LIN {X 0.059,Y -516.813,Z 888.156,A 0.000,B 0.000,C 90.000,E1 244.076} C_DIS
LIN {X -0.130,Y -514.887,Z 888.150,A 0.000,B 0.000,C 90.000,E1 242.922} C_DIS
LIN {X 0.096,Y -511.834,Z 888.140,A 0.000,B 0.000,C 90.000,E1 241.129} C_DIS
LIN {X -0.073,Y -508.198,Z 888.128,A 0.000,B 0.000,C 90.000,E1 239.076} C_DIS
LIN {X -0.008,Y -505.549,Z 888.120,A 0.000,B 0.000,C 90.000,E1 237.582} C_DIS
LIN {X 0.121,Y -503.196,Z 888.113,A 0.000,B 0.000,C 90.000,E1 236.373} C_DIS
LIN {X 0.071,Y -500.604,Z 888.107,A 0.000,B 0.000,C 90.000,E1 235.182} C_DIS
LIN {X -0.143,Y -497.089,Z 888.098,A 0.000,B 0.000,C 90.000,E1 233.703} C_DIS
LIN {X -0.267,Y -492.998,Z 888.088,A 0.000,B 0.000,C 90.000,E1 231.904} C_DIS
LIN {X -0.022,Y -489.498,Z 888.080,A 0.000,B 0.000,C 90.000,E1 230.356} C_DIS
LIN {X -0.047,Y -486.776,Z 888.073,A 0.000,B 0.000,C 90.000,E1 229.138} C_DIS
LIN {X 0.031,Y -483.298,Z 888.065,A 0.000,B 0.000,C 90.000,E1 227.595} C_DIS
LIN {X 0.037,Y -479.932,Z 888.056,A 0.000,B 0.000,C 90.000,E1 226.053} C_DIS
LIN {X 0.072,Y -475.754,Z 888.046,A 0.000,B 0.000,C 90.000,E1 224.190} C_DIS
LIN {X 0.120,Y -470.811,Z 888.033,A 0.000,B 0.000,C 90.000,E1 222.000} C_DIS
LIN {X -0.181,Y -468.009,Z 888.026,A 0.000,B 0.000,C 90.000,E1 220.782} C_DIS
LIN {X -0.109,Y -464.634,Z 888.018,A 0.000,B 0.000,C 90.000,E1 219.197} C_DIS
LIN {X -0.036,Y -461.259,Z 888.009,A 0.000,B 0.000,C 90.000,E1 217.604} C_DIS
LIN {X 0.078,Y -457.223,Z 887.998,A 0.000,B 0.000,C 90.000,E1 215.678} C_DIS
LIN {X -0.169,Y -453.164,Z 887.988,A 0.000,B 0.000,C 90.000,E1 213.785} C_DIS
LIN {X -0.069,Y -448.359,Z 887.975,A 0.000,B 0.000,C 90.000,E1 211.514} C_DIS
LIN {X 0.187,Y -443.374,Z 887.962,A 0.000,B 0.000,C 90.000,E1 209.205} C_DIS
LIN {X 0.179,Y -440.544,Z 887.955,A 0.000,B 0.000,C 90.000,E1 207.897} C_DIS
LIN {X -0.049,Y -436.846,Z 887.946,A 0.000,B 0.000,C 90.000,E1 206.283} C_DIS
LIN {X 0.072,Y -432.648,Z 887.935,A 0.000,B 0.000,C 90.000,E1 204.283} C_DIS
LIN {X 0.103,Y -428.359,Z 887.924,A 0.000,B 0.000,C 90.000,E1 202.280} C_DIS
LIN {X -0.126,Y -425.591,Z 887.916,A 0.000,B 0.000,C 90.000,E1 200.972} C_DIS
LIN {X -0.012,Y -420.825,Z 887.903,A 0.000,B 0.000,C 90.000,E1 198.598} C_DIS
LIN {X 0.069,Y -416.672,Z 887.892,A 0.000,B 0.000,C 90.000,E1 196.551} C_DIS
LIN {X -0.022,Y -411.180,Z 887.877,A 0.000,B 0.000,C 90.000,E1 193.828} C_DIS
LIN {X -0.115,Y -407.915,Z 887.867,A 0.000,B 0.000,C 90.000,E1 192.119} C_DIS
LIN {X 0.027,Y -405.234,Z 887.860,A 0.000,B 0.000,C 90.000,E1 190.715} C_DIS
LIN {X 0.043,Y -401.029,Z 887.848,A 0.000,B 0.000,C 90.000,E1 188.624} C_DIS
LIN {X -0.103,Y -396.837,Z 887.836,A 0.000,B 0.000,C 90.000,E1 186.543} C_DIS
LIN {X -0.116,Y -392.391,Z 887.823,A 0.000,B 0.000,C 90.000,E1 184.073} C_DIS
LIN {X -0.042,Y -387.473,Z 887.805,A 0.000,B 0.000,C 90.000,E1 180.859} C_DIS
LIN {X -0.040,Y -385.346,Z 887.797,A 0.000,B 0.000,C 90.000,E1 179.427} C_DIS
LIN {X -0.175,Y -382.648,Z 887.787,A 0.000,B 0.000,C 90.000,E1 177.650} C_DIS
LIN {X 0.135,Y -380.360,Z 887.779,A 0.000,B 0.000,C 90.000,E1 176.159} C_DIS
LIN {X -0.136,Y -376.095,Z 887.761,A 0.000,B 0.000,C 90.000,E1 172.932} C_DIS
LIN {X -0.027,Y -375.411,Z 887.757,A 0.000,B 0.000,C 90.000,E1 172.186} C_DIS
LIN {X 0.012,Y -374.903,Z 887.751,A 0.000,B 0.000,C 90.000,E1 171.084} C_DIS
LIN {X -0.099,Y -374.936,Z 887.748,A 0.000,B 0.000,C 90.000,E1 170.735} C_DIS
LIN {X 0.158,Y -374.805,Z 887.746,A 0.000,B 0.000,C 90.000,E1 170.330} C_DIS
LIN {X -0.090,Y -375.176,Z 887.741,A 0.000,B 0.000,C 90.000,E1 169.454} C_DIS
LIN {X 0.147,Y -375.812,Z 887.738,A 0.000,B 0.000,C 90.000,E1 168.870} C_DIS
LIN {X -0.001,Y -377.105,Z 887.734,A 0.000,B 0.000,C 90.000,E1 168.173} C_DIS
LIN {X -0.125,Y -378.598,Z 887.731,A 0.000,B 0.000,C 90.000,E1 167.645} C_DIS
LIN {X 0.093,Y -381.115,Z 887.728,A 0.000,B 0.000,C 90.000,E1 166.992} C_DIS
LIN {X -0.115,Y -384.469,Z 887.725,A 0.000,B 0.000,C 90.000,E1 166.464} C_DIS
LIN {X -0.114,Y -385.784,Z 887.724,A 0.000,B 0.000,C 90.000,E1 166.284} C_DIS
LIN {X 0.161,Y -389.176,Z 887.722,A 0.000,B 0.000,C 90.000,E1 165.880} C_DIS
LIN {X 0.093,Y -392.070,Z 887.720,A 0.000,B 0.000,C 90.000,E1 165.644} C_DIS
LIN {X 0.128,Y -398.264,Z 887.718,A 0.000,B 0.000,C 90.000,E1 165.227} C_DIS
LIN {X 0.093,Y -408.630,Z 887.715,A 0.000,B 0.000,C 90.000,E1 164.629} C_DIS
LIN {X -0.160,Y -413.785,Z 887.713,A 0.000,B 0.000,C 90.000,E1 164.393} C_DIS
LIN {X 0.051,Y -420.215,Z 887.711,A 0.000,B 0.000,C 90.000,E1 163.976} C_DIS
LIN {X -0.171,Y -429.850,Z 887.708,A 0.000,B 0.000,C 90.000,E1 163.378} C_DIS
LIN {X 0.016,Y -437.695,Z 887.704,A 0.000,B 0.000,C 90.000,E1 162.779} C_DIS
LIN {X 0.110,Y -446.755,Z 887.700,A 0.000,B 0.000,C 90.000,E1 162.000} C_DIS
LIN {X -0.047,Y -455.747,Z 887.696,A 0.000,B 0.000,C 90.000,E1 161.221} C_DIS
LIN {X 0.161,Y -464.336,Z 887.691,A 0.000,B 0.000,C 90.000,E1 160.369} C_DIS
LIN {X -0.030,Y -474.098,Z 887.686,A 0.000,B 0.000,C 90.000,E1 159.390} C_DIS
LIN {X 0.276,Y -481.913,Z 887.681,A 0.000,B 0.000,C 90.000,E1 158.465} C_DIS
LIN {X 0.065,Y -488.271,Z 887.676,A 0.000,B 0.000,C 90.000,E1 157.720} C_DIS
LIN {X 0.019,Y -499.849,Z 887.668,A 0.000,B 0.000,C 90.000,E1 156.230} C_DIS
LIN {X 0.044,Y -507.400,Z 887.662,A 0.000,B 0.000,C 90.000,E1 155.177} C_DIS
LIN {X 0.168,Y -510.575,Z 887.660,A 0.000,B 0.000,C 90.000,E1 154.717} C_DIS
LIN {X 0.050,Y -520.770,Z 887.651,A 0.000,B 0.000,C 90.000,E1 153.256} C_DIS
LIN {X -0.060,Y -528.491,Z 887.645,A 0.000,B 0.000,C 90.000,E1 152.103} C_DIS
LIN {X -0.099,Y -532.886,Z 887.641,A 0.000,B 0.000,C 90.000,E1 151.385} C_DIS
LIN {X -0.075,Y -538.842,Z 887.635,A 0.000,B 0.000,C 90.000,E1 150.383} C_DIS
LIN {X 0.117,Y -542.172,Z 887.632,A 0.000,B 0.000,C 90.000,E1 149.793} C_DIS
LIN {X -0.025,Y -549.222,Z 887.625,A 0.000,B 0.000,C 90.000,E1 148.535} C_DIS
LIN {X 0.188,Y -558.365,Z 887.616,A 0.000,B 0.000,C 90.000,E1 146.834} C_DIS
LIN {X 0.019,Y -565.388,Z 887.608,A 0.000,B 0.000,C 90.000,E1 145.468} C_DIS
LIN {X -0.177,Y -572.023,Z 887.601,A 0.000,B 0.000,C 90.000,E1 144.116} C_DIS
LIN {X 0.053,Y -577.218,Z 887.595,A 0.000,B 0.000,C 90.000,E1 143.004} C_DIS
LIN {X 0.242,Y -582.184,Z 887.589,A 0.000,B 0.000,C 90.000,E1 141.904} C_DIS
LIN {X -0.320,Y -587.103,Z 887.583,A 0.000,B 0.000,C 90.000,E1 140.884} C_DIS
LIN {X -0.248,Y -592.947,Z 887.575,A 0.000,B 0.000,C 90.000,E1 139.542} C_DIS
LIN {X 0.098,Y -599.979,Z 887.566,A 0.000,B 0.000,C 90.000,E1 137.919} C_DIS
LIN {X 0.146,Y -604.823,Z 887.560,A 0.000,B 0.000,C 90.000,E1 136.863} C_DIS
LIN {X -0.135,Y -611.955,Z 887.552,A 0.000,B 0.000,C 90.000,E1 135.324} C_DIS
LIN {X 0.051,Y -616.652,Z 887.546,A 0.000,B 0.000,C 90.000,E1 134.271} C_DIS
LIN {X -0.130,Y -621.125,Z 887.540,A 0.000,B 0.000,C 90.000,E1 133.257} C_DIS
LIN {X 0.311,Y -624.469,Z 887.536,A 0.000,B 0.000,C 90.000,E1 132.447} C_DIS
LIN {X -0.315,Y -629.897,Z 887.529,A 0.000,B 0.000,C 90.000,E1 131.229} C_DIS
LIN {X 0.152,Y -634.049,Z 887.523,A 0.000,B 0.000,C 90.000,E1 130.172} C_DIS
LIN {X -0.220,Y -638.094,Z 887.518,A 0.000,B 0.000,C 90.000,E1 129.197} C_DIS
LIN {X -0.147,Y -642.973,Z 887.511,A 0.000,B 0.000,C 90.000,E1 127.935} C_DIS
LIN {X 0.124,Y -647.825,Z 887.504,A 0.000,B 0.000,C 90.000,E1 126.664} C_DIS
LIN {X -0.044,Y -652.278,Z 887.497,A 0.000,B 0.000,C 90.000,E1 125.438} C_DIS
LIN {X 0.012,Y -656.493,Z 887.490,A 0.000,B 0.000,C 90.000,E1 124.199} C_DIS
LIN {X 0.144,Y -660.355,Z 887.483,A 0.000,B 0.000,C 90.000,E1 122.959} C_DIS
LIN {X 0.292,Y -662.401,Z 887.479,A 0.000,B 0.000,C 90.000,E1 122.212} C_DIS
LIN {X -0.105,Y -664.263,Z 887.475,A 0.000,B 0.000,C 90.000,E1 121.514} C_DIS
LIN {X -0.269,Y -665.852,Z 887.471,A 0.000,B 0.000,C 90.000,E1 120.797} C_DIS
LIN {X 0.075,Y -667.726,Z 887.466,A 0.000,B 0.000,C 90.000,E1 119.795} C_DIS
LIN {X -0.315,Y -669.714,Z 887.459,A 0.000,B 0.000,C 90.000,E1 118.615} C_DIS
LIN {X 0.256,Y -672.187,Z 887.449,A 0.000,B 0.000,C 90.000,E1 116.873} C_DIS
LIN {X 0.229,Y -673.346,Z 887.443,A 0.000,B 0.000,C 90.000,E1 115.668} C_DIS
LIN {X 0.150,Y -673.803,Z 887.439,A 0.000,B 0.000,C 90.000,E1 114.951} C_DIS
LIN {X -0.214,Y -674.045,Z 887.435,A 0.000,B 0.000,C 90.000,E1 114.259} C_DIS
LIN {X 0.041,Y -673.732,Z 887.431,A 0.000,B 0.000,C 90.000,E1 113.515} C_DIS
LIN {X 0.123,Y -672.857,Z 887.428,A 0.000,B 0.000,C 90.000,E1 113.025} C_DIS
LIN {X 0.294,Y -672.227,Z 887.427,A 0.000,B 0.000,C 90.000,E1 112.770} C_DIS
LIN {X -0.252,Y -669.397,Z 887.424,A 0.000,B 0.000,C 90.000,E1 112.333} C_DIS
LIN {X -0.172,Y -668.607,Z 887.423,A 0.000,B 0.000,C 90.000,E1 112.206} C_DIS
LIN {X -0.094,Y -667.531,Z 887.423,A 0.000,B 0.000,C 90.000,E1 112.078} C_DIS
LIN {X -0.171,Y -661.427,Z 887.420,A 0.000,B 0.000,C 90.000,E1 111.642} C_DIS
LIN {X -0.005,Y -659.918,Z 887.420,A 0.000,B 0.000,C 90.000,E1 111.535} C_DIS
LIN {X 0.346,Y -654.136,Z 887.418,A 0.000,B 0.000,C 90.000,E1 111.280} C_DIS
LIN {X 0.188,Y -652.034,Z 887.418,A 0.000,B 0.000,C 90.000,E1 111.227} C_DIS
LIN {X 0.362,Y -642.512,Z 887.417,A 0.000,B 0.000,C 90.000,E1 110.972} C_DIS
LIN {X -0.032,Y -634.972,Z 887.416,A 0.000,B 0.000,C 90.000,E1 110.844} C_DIS
LIN {X 0.254,Y -621.767,Z 887.414,A 0.000,B 0.000,C 90.000,E1 110.482} C_DIS
LIN {X 0.219,Y -615.744,Z 887.413,A 0.000,B 0.000,C 90.000,E1 110.301} C_DIS
LIN {X -0.145,Y -611.117,Z 887.412,A 0.000,B 0.000,C 90.000,E1 110.174} C_DIS
LIN {X 0.025,Y -603.066,Z 887.410,A 0.000,B 0.000,C 90.000,E1 109.812} C_DIS
LIN {X 0.054,Y -591.318,Z 887.407,A 0.000,B 0.000,C 90.000,E1 109.214} C_DIS
LIN {X 0.166,Y -588.091,Z 887.406,A 0.000,B 0.000,C 90.000,E1 109.033} C_DIS
LIN {X -0.159,Y -579.718,Z 887.404,A 0.000,B 0.000,C 90.000,E1 108.671} C_DIS
LIN {X -0.140,Y -567.602,Z 887.401,A 0.000,B 0.000,C 90.000,E1 108.236} C_DIS
LIN {X -0.094,Y -564.043,Z 887.401,A 0.000,B 0.000,C 90.000,E1 108.109} C_DIS
LIN {X 0.096,Y -562.050,Z 887.400,A 0.000,B 0.000,C 90.000,E1 108.000} C_DIS
LIN {X -0.011,Y -558.885,Z 887.399,A 0.000,B 0.000,C 90.000,E1 107.819} C_DIS
LIN {X -0.056,Y -558.823,Z 887.399,A 0.000,B 0.000,C 90.000,E1 107.819} C_DIS
LIN {X -0.160,Y -557.401,Z 887.398,A 0.000,B 0.000,C 90.000,E1 107.583} C_DIS
LIN {X -0.182,Y -556.754,Z 887.396,A 0.000,B 0.000,C 90.000,E1 107.221} C_DIS
LIN {X 0.149,Y -556.647,Z 887.391,A 0.000,B 0.000,C 90.000,E1 106.441} C_DIS
LIN {X 0.009,Y -557.505,Z 887.378,A 0.000,B 0.000,C 90.000,E1 103.953} C_DIS
LIN {X -0.235,Y -558.913,Z 887.364,A 0.000,B 0.000,C 90.000,E1 101.478} C_DIS
LIN {X 0.137,Y -560.336,Z 887.353,A 0.000,B 0.000,C 90.000,E1 99.500} C_DIS
LIN {X 0.239,Y -561.270,Z 887.345,A 0.000,B 0.000,C 90.000,E1 98.106} C_DIS
LIN {X -0.137,Y -562.309,Z 887.336,A 0.000,B 0.000,C 90.000,E1 96.486} C_DIS
LIN {X -0.237,Y -562.889,Z 887.330,A 0.000,B 0.000,C 90.000,E1 95.391} C_DIS
LIN {X -0.237,Y -563.548,Z 887.322,A 0.000,B 0.000,C 90.000,E1 94.012} C_DIS
LIN {X -0.261,Y -564.051,Z 887.315,A 0.000,B 0.000,C 90.000,E1 92.636} C_DIS
LIN {X -0.165,Y -564.603,Z 887.305,A 0.000,B 0.000,C 90.000,E1 90.974} C_DIS
LIN {X -0.067,Y -565.013,Z 887.296,A 0.000,B 0.000,C 90.000,E1 89.312} C_DIS
LIN {X -0.191,Y -565.269,Z 887.290,A 0.000,B 0.000,C 90.000,E1 88.224} C_DIS
LIN {X -0.156,Y -565.489,Z 887.282,A 0.000,B 0.000,C 90.000,E1 86.846} C_DIS
LIN {X 0.009,Y -565.757,Z 887.273,A 0.000,B 0.000,C 90.000,E1 85.179} C_DIS
LIN {X -0.142,Y -566.155,Z 887.261,A 0.000,B 0.000,C 90.000,E1 82.996} C_DIS
LIN {X -0.252,Y -566.636,Z 887.250,A 0.000,B 0.000,C 90.000,E1 81.084} C_DIS
LIN {X -0.249,Y -567.367,Z 887.240,A 0.000,B 0.000,C 90.000,E1 79.162} C_DIS
LIN {X -0.112,Y -568.261,Z 887.229,A 0.000,B 0.000,C 90.000,E1 77.229} C_DIS
LIN {X -0.006,Y -568.993,Z 887.220,A 0.000,B 0.000,C 90.000,E1 75.574} C_DIS
LIN {X 0.110,Y -569.714,Z 887.211,A 0.000,B 0.000,C 90.000,E1 73.921} C_DIS
LIN {X 0.179,Y -570.234,Z 887.200,A 0.000,B 0.000,C 90.000,E1 72.000} C_DIS
LIN {X -0.259,Y -570.502,Z 887.193,A 0.000,B 0.000,C 90.000,E1 70.678} C_DIS
LIN {X 0.059,Y -570.671,Z 887.188,A 0.000,B 0.000,C 90.000,E1 69.826} C_DIS
LIN {X -0.020,Y -570.836,Z 887.177,A 0.000,B 0.000,C 90.000,E1 67.922} C_DIS
LIN {X 0.167,Y -570.974,Z 887.170,A 0.000,B 0.000,C 90.000,E1 66.538} C_DIS
LIN {X -0.043,Y -570.967,Z 887.161,A 0.000,B 0.000,C 90.000,E1 64.921} C_DIS
LIN {X 0.227,Y -570.910,Z 887.152,A 0.000,B 0.000,C 90.000,E1 63.256} C_DIS
LIN {X -0.012,Y -570.603,Z 887.143,A 0.000,B 0.000,C 90.000,E1 61.641} C_DIS
LIN {X 0.187,Y -570.303,Z 887.135,A 0.000,B 0.000,C 90.000,E1 60.255} C_DIS
LIN {X -0.160,Y -570.175,Z 887.132,A 0.000,B 0.000,C 90.000,E1 59.744} C_DIS
LIN {X 0.134,Y -569.278,Z 887.123,A 0.000,B 0.000,C 90.000,E1 58.074} C_DIS
LIN {X 0.065,Y -569.010,Z 887.120,A 0.000,B 0.000,C 90.000,E1 57.533} C_DIS
LIN {X 0.233,Y -568.153,Z 887.114,A 0.000,B 0.000,C 90.000,E1 56.421} C_DIS
LIN {X 0.072,Y -567.176,Z 887.108,A 0.000,B 0.000,C 90.000,E1 55.341} C_DIS
LIN {X -0.249,Y -566.038,Z 887.101,A 0.000,B 0.000,C 90.000,E1 54.276} C_DIS
LIN {X 0.209,Y -564.558,Z 887.095,A 0.000,B 0.000,C 90.000,E1 53.130} C_DIS
LIN {X 0.091,Y -563.392,Z 887.091,A 0.000,B 0.000,C 90.000,E1 52.316} C_DIS
LIN {X 0.059,Y -562.076,Z 887.086,A 0.000,B 0.000,C 90.000,E1 51.492} C_DIS
LIN {X -0.086,Y -560.550,Z 887.082,A 0.000,B 0.000,C 90.000,E1 50.678} C_DIS
LIN {X 0.114,Y -558.831,Z 887.077,A 0.000,B 0.000,C 90.000,E1 49.828} C_DIS
LIN {X -0.141,Y -557.534,Z 887.074,A 0.000,B 0.000,C 90.000,E1 49.299} C_DIS
LIN {X 0.036,Y -555.312,Z 887.069,A 0.000,B 0.000,C 90.000,E1 48.447} C_DIS
LIN {X -0.181,Y -552.730,Z 887.065,A 0.000,B 0.000,C 90.000,E1 47.634} C_DIS
LIN {X -0.059,Y -549.844,Z 887.060,A 0.000,B 0.000,C 90.000,E1 46.782} C_DIS
LIN {X -0.365,Y -546.736,Z 887.055,A 0.000,B 0.000,C 90.000,E1 45.972} C_DIS
LIN {X 0.061,Y -544.472,Z 887.052,A 0.000,B 0.000,C 90.000,E1 45.364} C_DIS
LIN {X 0.268,Y -542.728,Z 887.050,A 0.000,B 0.000,C 90.000,E1 44.919} C_DIS
LIN {X -0.302,Y -539.400,Z 887.046,A 0.000,B 0.000,C 90.000,E1 44.271} C_DIS
LIN {X 0.067,Y -536.531,Z 887.043,A 0.000,B 0.000,C 90.000,E1 43.662} C_DIS
LIN {X 0.200,Y -532.521,Z 887.039,A 0.000,B 0.000,C 90.000,E1 42.933} C_DIS
LIN {X -0.064,Y -528.181,Z 887.035,A 0.000,B 0.000,C 90.000,E1 42.243} C_DIS
LIN {X -0.211,Y -522.699,Z 887.030,A 0.000,B 0.000,C 90.000,E1 41.391} C_DIS
LIN {X 0.111,Y -515.454,Z 887.024,A 0.000,B 0.000,C 90.000,E1 40.334} C_DIS
LIN {X -0.300,Y -509.888,Z 887.020,A 0.000,B 0.000,C 90.000,E1 39.644} C_DIS
LIN {X -0.051,Y -503.734,Z 887.016,A 0.000,B 0.000,C 90.000,E1 38.874} C_DIS
LIN {X 0.023,Y -499.850,Z 887.013,A 0.000,B 0.000,C 90.000,E1 38.418} C_DIS
LIN {X 0.121,Y -495.848,Z 887.011,A 0.000,B 0.000,C 90.000,E1 37.971} C_DIS
LIN {X -0.254,Y -490.285,Z 887.008,A 0.000,B 0.000,C 90.000,E1 37.443} C_DIS
LIN {X 0.038,Y -483.201,Z 887.004,A 0.000,B 0.000,C 90.000,E1 36.710} C_DIS
LIN {X 0.255,Y -475.862,Z 887.000,A 0.000,B 0.000,C 90.000,E1 36.011} C_DIS
LIN {X -0.122,Y -465.301,Z 886.995,A 0.000,B 0.000,C 90.000,E1 35.152} C_DIS
LIN {X -0.131,Y -454.806,Z 886.990,A 0.000,B 0.000,C 90.000,E1 34.278} C_DIS
LIN {X 0.057,Y -437.675,Z 886.983,A 0.000,B 0.000,C 90.000,E1 32.880} C_DIS
LIN {X 0.055,Y -416.158,Z 886.973,A 0.000,B 0.000,C 90.000,E1 31.052} C_DIS
LIN {X -0.042,Y -402.686,Z 886.966,A 0.000,B 0.000,C 90.000,E1 29.795} C_DIS
LIN {X 0.018,Y -398.395,Z 886.963,A 0.000,B 0.000,C 90.000,E1 29.333} C_DIS
LIN {X -0.224,Y -394.895,Z 886.961,A 0.000,B 0.000,C 90.000,E1 28.949} C_DIS
LIN {X -0.097,Y -391.850,Z 886.958,A 0.000,B 0.000,C 90.000,E1 28.409} C_DIS
LIN {X 0.110,Y -390.090,Z 886.955,A 0.000,B 0.000,C 90.000,E1 27.847} C_DIS
LIN {X 0.148,Y -389.174,Z 886.951,A 0.000,B 0.000,C 90.000,E1 27.129} C_DIS
LIN {X 0.182,Y -389.082,Z 886.946,A 0.000,B 0.000,C 90.000,E1 26.232} C_DIS
LIN {X 0.056,Y -389.793,Z 886.938,A 0.000,B 0.000,C 90.000,E1 24.823} C_DIS
LIN {X 0.036,Y -391.867,Z 886.924,A 0.000,B 0.000,C 90.000,E1 22.333} C_DIS
LIN {X -0.018,Y -394.747,Z 886.908,A 0.000,B 0.000,C 90.000,E1 19.504} C_DIS
LIN {X -0.067,Y -397.577,Z 886.895,A 0.000,B 0.000,C 90.000,E1 17.040} C_DIS
LIN {X -0.150,Y -400.720,Z 886.881,A 0.000,B 0.000,C 90.000,E1 14.592} C_DIS
LIN {X 0.038,Y -405.029,Z 886.864,A 0.000,B 0.000,C 90.000,E1 11.422} C_DIS
LIN {X 0.158,Y -407.697,Z 886.854,A 0.000,B 0.000,C 90.000,E1 9.670} C_DIS
LIN {X -0.155,Y -411.645,Z 886.840,A 0.000,B 0.000,C 90.000,E1 7.296} C_DIS
LIN {X 0.000,Y -416.709,Z 886.825,A 0.000,B 0.000,C 90.000,E1 4.531} C_DIS
LIN {X -0.089,Y -423.732,Z 886.806,A 0.000,B 0.000,C 90.000,E1 1.146} C_DIS
LIN {X -0.081,Y -429.251,Z 886.793,A 0.000,B 0.000,C 90.000,E1 358.797} C_DIS
LIN {X 0.145,Y -436.063,Z 886.779,A 0.000,B 0.000,C 90.000,E1 356.102} C_DIS
LIN {X -0.077,Y -438.183,Z 886.775,A 0.000,B 0.000,C 90.000,E1 355.469} C_DIS
LIN {X 0.055,Y -439.675,Z 886.773,A 0.000,B 0.000,C 90.000,E1 355.122} C_DIS
LIN {X 0.001,Y -442.807,Z 886.770,A 0.000,B 0.000,C 90.000,E1 354.609} C_DIS
LIN {X -0.192,Y -443.523,Z 886.770,A 0.000,B 0.000,C 90.000,E1 354.546} C_DIS
LIN {X 0.015,Y -444.471,Z 886.769,A 0.000,B 0.000,C 90.000,E1 354.432} C_DIS
LIN {X -0.016,Y -449.205,Z 886.767,A 0.000,B 0.000,C 90.000,E1 354.090} C_DIS
LIN {X 0.103,Y -456.288,Z 886.765,A 0.000,B 0.000,C 90.000,E1 353.742} C_DIS
LIN {X -0.076,Y -468.575,Z 886.762,A 0.000,B 0.000,C 90.000,E1 353.223} C_DIS
LIN {X 0.223,Y -475.053,Z 886.761,A 0.000,B 0.000,C 90.000,E1 352.875} C_DIS
LIN {X 0.208,Y -481.798,Z 886.759,A 0.000,B 0.000,C 90.000,E1 352.534} C_DIS
LIN {X 0.135,Y -491.540,Z 886.756,A 0.000,B 0.000,C 90.000,E1 352.008} C_DIS
LIN {X 0.171,Y -501.419,Z 886.753,A 0.000,B 0.000,C 90.000,E1 351.432} C_DIS
LIN {X -0.122,Y -513.963,Z 886.748,A 0.000,B 0.000,C 90.000,E1 350.679} C_DIS
LIN {X -0.079,Y -521.715,Z 886.745,A 0.000,B 0.000,C 90.000,E1 350.151} C_DIS
LIN {X 0.198,Y -529.264,Z 886.742,A 0.000,B 0.000,C 90.000,E1 349.577} C_DIS
LIN {X -0.223,Y -538.117,Z 886.738,A 0.000,B 0.000,C 90.000,E1 348.926} C_DIS
LIN {X 0.153,Y -543.635,Z 886.736,A 0.000,B 0.000,C 90.000,E1 348.409} C_DIS
LIN {X -0.136,Y -549.131,Z 886.733,A 0.000,B 0.000,C 90.000,E1 347.937} C_DIS
LIN {X -0.033,Y -554.512,Z 886.730,A 0.000,B 0.000,C 90.000,E1 347.409} C_DIS
LIN {X -0.159,Y -560.835,Z 886.726,A 0.000,B 0.000,C 90.000,E1 346.756} C_DIS
LIN {X -0.069,Y -566.929,Z 886.723,A 0.000,B 0.000,C 90.000,E1 346.061} C_DIS
LIN {X -0.139,Y -571.537,Z 886.720,A 0.000,B 0.000,C 90.000,E1 345.519} C_DIS
LIN {X -0.121,Y -577.964,Z 886.715,A 0.000,B 0.000,C 90.000,E1 344.700} C_DIS
LIN {X 0.114,Y -583.849,Z 886.710,A 0.000,B 0.000,C 90.000,E1 343.866} C_DIS
LIN {X -0.150,Y -589.341,Z 886.706,A 0.000,B 0.000,C 90.000,E1 343.087} C_DIS
LIN {X 0.021,Y -596.755,Z 886.699,A 0.000,B 0.000,C 90.000,E1 341.873} C_DIS
LIN {X -0.111,Y -601.276,Z 886.695,A 0.000,B 0.000,C 90.000,E1 341.094} C_DIS
LIN {X -0.247,Y -606.318,Z 886.690,A 0.000,B 0.000,C 90.000,E1 340.188} C_DIS
LIN {X -0.384,Y -612.346,Z 886.683,A 0.000,B 0.000,C 90.000,E1 339.028} C_DIS
LIN {X -0.178,Y -616.855,Z 886.678,A 0.000,B 0.000,C 90.000,E1 338.103} C_DIS
LIN {X 0.078,Y -621.677,Z 886.673,A 0.000,B 0.000,C 90.000,E1 337.050} C_DIS
LIN {X -0.181,Y -626.221,Z 886.667,A 0.000,B 0.000,C 90.000,E1 336.049} C_DIS
LIN {X -0.120,Y -630.452,Z 886.661,A 0.000,B 0.000,C 90.000,E1 335.025} C_DIS
LIN {X -0.267,Y -634.393,Z 886.656,A 0.000,B 0.000,C 90.000,E1 334.024} C_DIS
LIN {X -0.090,Y -638.035,Z 886.650,A 0.000,B 0.000,C 90.000,E1 332.999} C_DIS
LIN {X 0.017,Y -639.804,Z 886.647,A 0.000,B 0.000,C 90.000,E1 332.487} C_DIS
LIN {X -0.303,Y -643.095,Z 886.642,A 0.000,B 0.000,C 90.000,E1 331.513} C_DIS
LIN {X 0.295,Y -646.090,Z 886.636,A 0.000,B 0.000,C 90.000,E1 330.461} C_DIS
LIN {X 0.048,Y -649.045,Z 886.631,A 0.000,B 0.000,C 90.000,E1 329.488} C_DIS
LIN {X 0.039,Y -652.487,Z 886.624,A 0.000,B 0.000,C 90.000,E1 328.250} C_DIS
LIN {X -0.241,Y -654.411,Z 886.620,A 0.000,B 0.000,C 90.000,E1 327.533} C_DIS
LIN {X -0.155,Y -657.153,Z 886.613,A 0.000,B 0.000,C 90.000,E1 326.294} C_DIS
LIN {X -0.119,Y -659.133,Z 886.607,A 0.000,B 0.000,C 90.000,E1 325.308} C_DIS
LIN {X 0.042,Y -661.153,Z 886.600,A 0.000,B 0.000,C 90.000,E1 324.069} C_DIS
LIN {X -0.404,Y -662.539,Z 886.595,A 0.000,B 0.000,C 90.000,E1 323.130} C_DIS
LIN {X 0.102,Y -663.796,Z 886.590,A 0.000,B 0.000,C 90.000,E1 322.110} C_DIS
LIN {X 0.188,Y -665.124,Z 886.583,A 0.000,B 0.000,C 90.000,E1 320.884} C_DIS
LIN {X 0.249,Y -667.167,Z 886.572,A 0.000,B 0.000,C 90.000,E1 318.933} C_DIS
LIN {X 0.302,Y -668.974,Z 886.563,A 0.000,B 0.000,C 90.000,E1 317.229} C_DIS
LIN {X -0.104,Y -670.500,Z 886.555,A 0.000,B 0.000,C 90.000,E1 315.810} C_DIS
LIN {X -0.015,Y -671.971,Z 886.546,A 0.000,B 0.000,C 90.000,E1 314.352} C_DIS
LIN {X -0.324,Y -673.867,Z 886.536,A 0.000,B 0.000,C 90.000,E1 312.447} C_DIS
LIN {X -0.168,Y -674.987,Z 886.529,A 0.000,B 0.000,C 90.000,E1 311.229} C_DIS
LIN {X 0.155,Y -676.657,Z 886.518,A 0.000,B 0.000,C 90.000,E1 309.277} C_DIS
LIN {X -0.078,Y -677.578,Z 886.512,A 0.000,B 0.000,C 90.000,E1 308.096} C_DIS
LIN {X 0.235,Y -678.498,Z 886.505,A 0.000,B 0.000,C 90.000,E1 306.870} C_DIS
LIN {X 0.164,Y -679.304,Z 886.498,A 0.000,B 0.000,C 90.000,E1 305.678} C_DIS
LIN {X 0.108,Y -680.035,Z 886.492,A 0.000,B 0.000,C 90.000,E1 304.485} C_DIS
LIN {X 0.409,Y -681.239,Z 886.481,A 0.000,B 0.000,C 90.000,E1 302.546} C_DIS
LIN {X 0.004,Y -682.660,Z 886.470,A 0.000,B 0.000,C 90.000,E1 300.669} C_DIS
LIN {X 0.009,Y -684.099,Z 886.461,A 0.000,B 0.000,C 90.000,E1 298.999} C_DIS
LIN {X 0.211,Y -686.165,Z 886.451,A 0.000,B 0.000,C 90.000,E1 297.078} C_DIS
LIN {X -0.142,Y -688.455,Z 886.440,A 0.000,B 0.000,C 90.000,E1 295.207} C_DIS
LIN {X -0.194,Y -689.561,Z 886.433,A 0.000,B 0.000,C 90.000,E1 294.027} C_DIS
LIN {X 0.268,Y -689.916,Z 886.431,A 0.000,B 0.000,C 90.000,E1 293.515} C_DIS
LIN {X -0.408,Y -689.929,Z 886.430,A 0.000,B 0.000,C 90.000,E1 293.334} C_DIS
LIN {X 0.051,Y -689.678,Z 886.427,A 0.000,B 0.000,C 90.000,E1 292.823} C_DIS
LIN {X 0.013,Y -689.142,Z 886.426,A 0.000,B 0.000,C 90.000,E1 292.589} C_DIS
LIN {X 0.204,Y -687.622,Z 886.423,A 0.000,B 0.000,C 90.000,E1 292.099} C_DIS
LIN {X -0.323,Y -686.971,Z 886.422,A 0.000,B 0.000,C 90.000,E1 292.025} C_DIS
LIN {X -0.212,Y -685.996,Z 886.422,A 0.000,B 0.000,C 90.000,E1 291.897} C_DIS
LIN {X 0.001,Y -683.493,Z 886.420,A 0.000,B 0.000,C 90.000,E1 291.642} C_DIS
LIN {X 0.104,Y -680.957,Z 886.419,A 0.000,B 0.000,C 90.000,E1 291.408} C_DIS
LIN {X 0.282,Y -679.253,Z 886.418,A 0.000,B 0.000,C 90.000,E1 291.280} C_DIS
LIN {X 0.213,Y -676.257,Z 886.418,A 0.000,B 0.000,C 90.000,E1 291.173} C_DIS
LIN {X -0.184,Y -669.080,Z 886.416,A 0.000,B 0.000,C 90.000,E1 290.972} C_DIS
LIN {X 0.061,Y -661.537,Z 886.415,A 0.000,B 0.000,C 90.000,E1 290.737} C_DIS
LIN {X -0.183,Y -656.899,Z 886.414,A 0.000,B 0.000,C 90.000,E1 290.536} C_DIS
LIN {X 0.374,Y -656.815,Z 886.414,A 0.000,B 0.000,C 90.000,E1 290.482} C_DIS
LIN {X -0.016,Y -655.833,Z 886.413,A 0.000,B 0.000,C 90.000,E1 290.375} C_DIS
LIN {X -0.060,Y -655.822,Z 886.413,A 0.000,B 0.000,C 90.000,E1 290.375} C_DIS
LIN {X -0.046,Y -655.737,Z 886.412,A 0.000,B 0.000,C 90.000,E1 290.174} C_DIS
LIN {X -0.077,Y -657.252,Z 886.409,A 0.000,B 0.000,C 90.000,E1 289.685} C_DIS
LIN {X -0.209,Y -660.425,Z 886.406,A 0.000,B 0.000,C 90.000,E1 289.033} C_DIS
LIN {X -0.201,Y -664.986,Z 886.401,A 0.000,B 0.000,C 90.000,E1 288.181} C_DIS
LIN {X -0.236,Y -666.887,Z 886.399,A 0.000,B 0.000,C 90.000,E1 287.819} C_DIS
LIN {X -0.285,Y -670.305,Z 886.395,A 0.000,B 0.000,C 90.000,E1 287.094} C_DIS
LIN {X 0.214,Y -672.292,Z 886.392,A 0.000,B 0.000,C 90.000,E1 286.567} C_DIS
LIN {X 0.216,Y -674.817,Z 886.388,A 0.000,B 0.000,C 90.000,E1 285.843} C_DIS
LIN {X 0.055,Y -676.701,Z 886.384,A 0.000,B 0.000,C 90.000,E1 285.134} C_DIS
LIN {X -0.040,Y -677.804,Z 886.381,A 0.000,B 0.000,C 90.000,E1 284.662} C_DIS
LIN {X -0.004,Y -679.141,Z 886.378,A 0.000,B 0.000,C 90.000,E1 283.939} C_DIS
LIN {X -0.282,Y -680.271,Z 886.373,A 0.000,B 0.000,C 90.000,E1 283.244} C_DIS
LIN {X 0.276,Y -681.127,Z 886.370,A 0.000,B 0.000,C 90.000,E1 282.479} C_DIS
LIN {X 0.173,Y -681.667,Z 886.366,A 0.000,B 0.000,C 90.000,E1 281.771} C_DIS
LIN {X 0.103,Y -681.830,Z 886.363,A 0.000,B 0.000,C 90.000,E1 281.299} C_DIS
LIN {X -0.133,Y -681.447,Z 886.359,A 0.000,B 0.000,C 90.000,E1 280.602} C_DIS
LIN {X -0.330,Y -680.970,Z 886.356,A 0.000,B 0.000,C 90.000,E1 280.141} C_DIS
LIN {X 0.261,Y -680.172,Z 886.354,A 0.000,B 0.000,C 90.000,E1 279.613} C_DIS
LIN {X 0.060,Y -679.042,Z 886.351,A 0.000,B 0.000,C 90.000,E1 279.151} C_DIS
LIN {X -0.195,Y -676.772,Z 886.347,A 0.000,B 0.000,C 90.000,E1 278.454} C_DIS
LIN {X 0.259,Y -674.965,Z 886.344,A 0.000,B 0.000,C 90.000,E1 277.936} C_DIS
LIN {X 0.035,Y -672.807,Z 886.342,A 0.000,B 0.000,C 90.000,E1 277.473} C_DIS
LIN {X -0.201,Y -669.739,Z 886.338,A 0.000,B 0.000,C 90.000,E1 276.891} C_DIS
LIN {X 0.116,Y -666.230,Z 886.335,A 0.000,B 0.000,C 90.000,E1 276.258} C_DIS
LIN {X -0.167,Y -663.120,Z 886.332,A 0.000,B 0.000,C 90.000,E1 275.796} C_DIS
LIN {X 0.186,Y -659.553,Z 886.329,A 0.000,B 0.000,C 90.000,E1 275.277} C_DIS
LIN {X -0.196,Y -655.508,Z 886.327,A 0.000,B 0.000,C 90.000,E1 274.821} C_DIS
LIN {X 0.134,Y -649.860,Z 886.323,A 0.000,B 0.000,C 90.000,E1 274.188} C_DIS
LIN {X -0.004,Y -645.037,Z 886.321,A 0.000,B 0.000,C 90.000,E1 273.726} C_DIS
LIN {X -0.144,Y -638.427,Z 886.318,A 0.000,B 0.000,C 90.000,E1 273.154} C_DIS
LIN {X 0.024,Y -631.476,Z 886.314,A 0.000,B 0.000,C 90.000,E1 272.579} C_DIS
LIN {X -0.023,Y -623.963,Z 886.312,A 0.000,B 0.000,C 90.000,E1 272.064} C_DIS
LIN {X 0.152,Y -617.581,Z 886.309,A 0.000,B 0.000,C 90.000,E1 271.661} C_DIS
LIN {X 0.008,Y -611.071,Z 886.307,A 0.000,B 0.000,C 90.000,E1 271.318} C_DIS
LIN {X 0.093,Y -602.622,Z 886.305,A 0.000,B 0.000,C 90.000,E1 270.917} C_DIS
LIN {X 0.192,Y -597.525,Z 886.304,A 0.000,B 0.000,C 90.000,E1 270.688} C_DIS
LIN {X -0.232,Y -589.970,Z 886.302,A 0.000,B 0.000,C 90.000,E1 270.458} C_DIS
LIN {X -0.244,Y -584.419,Z 886.302,A 0.000,B 0.000,C 90.000,E1 270.286} C_DIS
LIN {X 0.062,Y -576.820,Z 886.300,A 0.000,B 0.000,C 90.000,E1 270.057} C_DIS
LIN {X 0.026,Y -570.829,Z 886.300,A 0.000,B 0.000,C 90.000,E1 269.943} C_DIS
LIN {X -0.119,Y -564.792,Z 886.299,A 0.000,B 0.000,C 90.000,E1 269.885} C_DIS
LIN {X 0.045,Y -552.116,Z 886.299,A 0.000,B 0.000,C 90.000,E1 269.771} C_DIS
LIN {X -0.037,Y -549.913,Z 886.298,A 0.000,B 0.000,C 90.000,E1 269.714} C_DIS
LIN {X -0.080,Y -549.791,Z 886.298,A 0.000,B 0.000,C 90.000,E1 269.714} C_DIS
LIN {X 0.052,Y -548.303,Z 886.298,A 0.000,B 0.000,C 90.000,E1 269.542} C_DIS
LIN {X 0.013,Y -546.367,Z 886.297,A 0.000,B 0.000,C 90.000,E1 269.370} C_DIS
LIN {X -0.026,Y -546.334,Z 886.297,A 0.000,B 0.000,C 90.000,E1 269.370} C_DIS
LIN {X 0.161,Y -545.150,Z 886.294,A 0.000,B 0.000,C 90.000,E1 268.854} C_DIS
LIN {X -0.137,Y -543.395,Z 886.286,A 0.000,B 0.000,C 90.000,E1 267.478} C_DIS
LIN {X 0.197,Y -541.262,Z 886.270,A 0.000,B 0.000,C 90.000,E1 264.609} C_DIS
LIN {X -0.130,Y -540.337,Z 886.262,A 0.000,B 0.000,C 90.000,E1 263.223} C_DIS
LIN {X 0.072,Y -539.410,Z 886.256,A 0.000,B 0.000,C 90.000,E1 262.064} C_DIS
LIN {X -0.287,Y -538.034,Z 886.248,A 0.000,B 0.000,C 90.000,E1 260.679} C_DIS
LIN {X 0.156,Y -535.947,Z 886.237,A 0.000,B 0.000,C 90.000,E1 258.634} C_DIS
LIN {X -0.081,Y -534.405,Z 886.229,A 0.000,B 0.000,C 90.000,E1 257.229} C_DIS
LIN {X -0.181,Y -532.235,Z 886.219,A 0.000,B 0.000,C 90.000,E1 255.519} C_DIS
LIN {X -0.195,Y -530.058,Z 886.210,A 0.000,B 0.000,C 90.000,E1 253.795} C_DIS
LIN {X -0.106,Y -528.026,Z 886.200,A 0.000,B 0.000,C 90.000,E1 252.054} C_DIS
LIN {X 0.083,Y -526.906,Z 886.195,A 0.000,B 0.000,C 90.000,E1 251.167} C_DIS
LIN {X -0.061,Y -524.711,Z 886.186,A 0.000,B 0.000,C 90.000,E1 249.444} C_DIS
LIN {X -0.075,Y -523.132,Z 886.179,A 0.000,B 0.000,C 90.000,E1 248.284} C_DIS
LIN {X 0.233,Y -521.027,Z 886.171,A 0.000,B 0.000,C 90.000,E1 246.794} C_DIS
LIN {X -0.121,Y -519.243,Z 886.165,A 0.000,B 0.000,C 90.000,E1 245.665} C_DIS
LIN {X -0.144,Y -517.037,Z 886.157,A 0.000,B 0.000,C 90.000,E1 244.204} C_DIS
LIN {X 0.007,Y -515.611,Z 886.152,A 0.000,B 0.000,C 90.000,E1 243.307} C_DIS
LIN {X -0.093,Y -513.057,Z 886.144,A 0.000,B 0.000,C 90.000,E1 241.847} C_DIS
LIN {X -0.105,Y -511.014,Z 886.137,A 0.000,B 0.000,C 90.000,E1 240.667} C_DIS
LIN {X -0.255,Y -508.458,Z 886.129,A 0.000,B 0.000,C 90.000,E1 239.203} C_DIS
LIN {X -0.076,Y -506.301,Z 886.122,A 0.000,B 0.000,C 90.000,E1 237.995} C_DIS
LIN {X -0.245,Y -504.636,Z 886.117,A 0.000,B 0.000,C 90.000,E1 237.120} C_DIS
LIN {X 0.028,Y -501.586,Z 886.109,A 0.000,B 0.000,C 90.000,E1 235.595} C_DIS
LIN {X -0.040,Y -498.826,Z 886.102,A 0.000,B 0.000,C 90.000,E1 234.402} C_DIS
LIN {X 0.270,Y -494.676,Z 886.092,A 0.000,B 0.000,C 90.000,E1 232.557} C_DIS
LIN {X -0.299,Y -490.500,Z 886.082,A 0.000,B 0.000,C 90.000,E1 230.803} C_DIS
LIN {X 0.040,Y -486.313,Z 886.072,A 0.000,B 0.000,C 90.000,E1 228.933} C_DIS
LIN {X -0.036,Y -483.549,Z 886.065,A 0.000,B 0.000,C 90.000,E1 227.715} C_DIS
LIN {X 0.299,Y -480.210,Z 886.057,A 0.000,B 0.000,C 90.000,E1 226.134} C_DIS
LIN {X -0.002,Y -476.069,Z 886.046,A 0.000,B 0.000,C 90.000,E1 224.312} C_DIS
LIN {X -0.187,Y -470.438,Z 886.032,A 0.000,B 0.000,C 90.000,E1 221.838} C_DIS
LIN {X 0.172,Y -464.930,Z 886.018,A 0.000,B 0.000,C 90.000,E1 219.277} C_DIS
LIN {X 0.000,Y -460.827,Z 886.008,A 0.000,B 0.000,C 90.000,E1 217.397} C_DIS
LIN {X 0.000,Y -457.518,Z 885.999,A 0.000,B 0.000,C 90.000,E1 215.804} C_DIS
LIN {X 0.132,Y -453.464,Z 885.988,A 0.000,B 0.000,C 90.000,E1 213.865} C_DIS
LIN {X 0.243,Y -448.641,Z 885.976,A 0.000,B 0.000,C 90.000,E1 211.592} C_DIS
LIN {X 0.062,Y -444.389,Z 885.965,A 0.000,B 0.000,C 90.000,E1 209.667} C_DIS
LIN {X 0.072,Y -441.636,Z 885.958,A 0.000,B 0.000,C 90.000,E1 208.359} C_DIS
LIN {X -0.129,Y -437.912,Z 885.949,A 0.000,B 0.000,C 90.000,E1 206.744} C_DIS
LIN {X 0.206,Y -432.995,Z 885.936,A 0.000,B 0.000,C 90.000,E1 204.387} C_DIS
LIN {X 0.069,Y -428.701,Z 885.925,A 0.000,B 0.000,C 90.000,E1 202.408} C_DIS
LIN {X 0.044,Y -425.230,Z 885.915,A 0.000,B 0.000,C 90.000,E1 200.737} C_DIS
LIN {X -0.023,Y -421.196,Z 885.904,A 0.000,B 0.000,C 90.000,E1 198.725} C_DIS
LIN {X 0.070,Y -417.026,Z 885.893,A 0.000,B 0.000,C 90.000,E1 196.677} C_DIS
LIN {X 0.000,Y -411.536,Z 885.878,A 0.000,B 0.000,C 90.000,E1 193.953} C_DIS
LIN {X 0.026,Y -407.599,Z 885.866,A 0.000,B 0.000,C 90.000,E1 191.883} C_DIS
LIN {X 0.085,Y -404.887,Z 885.858,A 0.000,B 0.000,C 90.000,E1 190.489} C_DIS
LIN {X 0.106,Y -401.408,Z 885.849,A 0.000,B 0.000,C 90.000,E1 188.746} C_DIS
LIN {X -0.020,Y -397.193,Z 885.837,A 0.000,B 0.000,C 90.000,E1 186.663} C_DIS
LIN {X -0.033,Y -392.114,Z 885.821,A 0.000,B 0.000,C 90.000,E1 183.841} C_DIS
LIN {X 0.008,Y -387.312,Z 885.804,A 0.000,B 0.000,C 90.000,E1 180.630} C_DIS
LIN {X 0.006,Y -385.134,Z 885.796,A 0.000,B 0.000,C 90.000,E1 179.198} C_DIS
LIN {X -0.134,Y -382.474,Z 885.786,A 0.000,B 0.000,C 90.000,E1 177.421} C_DIS
LIN {X -0.085,Y -380.779,Z 885.780,A 0.000,B 0.000,C 90.000,E1 176.331} C_DIS
LIN {X 0.152,Y -375.555,Z 885.757,A 0.000,B 0.000,C 90.000,E1 172.299} C_DIS
LIN {X 0.195,Y -374.826,Z 885.751,A 0.000,B 0.000,C 90.000,E1 171.197} C_DIS
LIN {X -0.028,Y -374.622,Z 885.747,A 0.000,B 0.000,C 90.000,E1 170.500} C_DIS
LIN {X 0.026,Y -374.697,Z 885.742,A 0.000,B 0.000,C 90.000,E1 169.577} C_DIS
LIN {X -0.074,Y -375.104,Z 885.740,A 0.000,B 0.000,C 90.000,E1 169.162} C_DIS
LIN {X 0.067,Y -375.648,Z 885.736,A 0.000,B 0.000,C 90.000,E1 168.409} C_DIS
LIN {X -0.080,Y -377.174,Z 885.732,A 0.000,B 0.000,C 90.000,E1 167.701} C_DIS
LIN {X 0.167,Y -378.930,Z 885.729,A 0.000,B 0.000,C 90.000,E1 167.117} C_DIS
LIN {X 0.054,Y -381.129,Z 885.726,A 0.000,B 0.000,C 90.000,E1 166.589} C_DIS
LIN {X -0.046,Y -384.164,Z 885.723,A 0.000,B 0.000,C 90.000,E1 166.061} C_DIS
LIN {X 0.008,Y -387.061,Z 885.721,A 0.000,B 0.000,C 90.000,E1 165.700} C_DIS
LIN {X 0.061,Y -388.697,Z 885.720,A 0.000,B 0.000,C 90.000,E1 165.519} C_DIS
LIN {X -0.115,Y -393.277,Z 885.718,A 0.000,B 0.000,C 90.000,E1 165.172} C_DIS
LIN {X -0.048,Y -396.630,Z 885.716,A 0.000,B 0.000,C 90.000,E1 164.936} C_DIS
LIN {X -0.195,Y -415.368,Z 885.711,A 0.000,B 0.000,C 90.000,E1 163.921} C_DIS
LIN {X -0.003,Y -421.885,Z 885.708,A 0.000,B 0.000,C 90.000,E1 163.504} C_DIS
LIN {X 0.013,Y -428.167,Z 885.706,A 0.000,B 0.000,C 90.000,E1 163.087} C_DIS
LIN {X 0.225,Y -437.799,Z 885.702,A 0.000,B 0.000,C 90.000,E1 162.362} C_DIS
LIN {X 0.069,Y -443.742,Z 885.700,A 0.000,B 0.000,C 90.000,E1 161.891} C_DIS
LIN {X 0.167,Y -452.824,Z 885.695,A 0.000,B 0.000,C 90.000,E1 161.094} C_DIS
LIN {X -0.140,Y -457.174,Z 885.693,A 0.000,B 0.000,C 90.000,E1 160.732} C_DIS
LIN {X 0.031,Y -464.383,Z 885.689,A 0.000,B 0.000,C 90.000,E1 160.007} C_DIS
LIN {X 0.289,Y -471.450,Z 885.685,A 0.000,B 0.000,C 90.000,E1 159.263} C_DIS
LIN {X 0.006,Y -479.510,Z 885.680,A 0.000,B 0.000,C 90.000,E1 158.411} C_DIS
LIN {X 0.124,Y -487.192,Z 885.675,A 0.000,B 0.000,C 90.000,E1 157.486} C_DIS
LIN {X -0.119,Y -494.266,Z 885.670,A 0.000,B 0.000,C 90.000,E1 156.613} C_DIS
LIN {X -0.103,Y -500.029,Z 885.666,A 0.000,B 0.000,C 90.000,E1 155.869} C_DIS
LIN {X 0.131,Y -507.638,Z 885.660,A 0.000,B 0.000,C 90.000,E1 154.793} C_DIS
LIN {X -0.153,Y -519.954,Z 885.650,A 0.000,B 0.000,C 90.000,E1 153.050} C_DIS
LIN {X -0.118,Y -526.732,Z 885.645,A 0.000,B 0.000,C 90.000,E1 152.025} C_DIS
LIN {X 0.109,Y -533.850,Z 885.638,A 0.000,B 0.000,C 90.000,E1 150.845} C_DIS
LIN {X -0.294,Y -540.571,Z 885.632,A 0.000,B 0.000,C 90.000,E1 149.744} C_DIS
LIN {X -0.185,Y -547.727,Z 885.625,A 0.000,B 0.000,C 90.000,E1 148.456} C_DIS
LIN {X -0.188,Y -556.262,Z 885.616,A 0.000,B 0.000,C 90.000,E1 146.914} C_DIS
LIN {X -0.290,Y -562.644,Z 885.609,A 0.000,B 0.000,C 90.000,E1 145.674} C_DIS
LIN {X -0.073,Y -569.406,Z 885.602,A 0.000,B 0.000,C 90.000,E1 144.276} C_DIS
LIN {X -0.200,Y -576.024,Z 885.594,A 0.000,B 0.000,C 90.000,E1 142.924} C_DIS
LIN {X 0.038,Y -584.780,Z 885.583,A 0.000,B 0.000,C 90.000,E1 141.009} C_DIS
LIN {X -0.011,Y -591.353,Z 885.575,A 0.000,B 0.000,C 90.000,E1 139.542} C_DIS
LIN {X -0.293,Y -594.805,Z 885.571,A 0.000,B 0.000,C 90.000,E1 138.771} C_DIS
LIN {X 0.014,Y -602.621,Z 885.561,A 0.000,B 0.000,C 90.000,E1 137.025} C_DIS
LIN {X 0.213,Y -609.278,Z 885.553,A 0.000,B 0.000,C 90.000,E1 135.567} C_DIS
LIN {X 0.197,Y -615.198,Z 885.546,A 0.000,B 0.000,C 90.000,E1 134.271} C_DIS
LIN {X -0.308,Y -621.980,Z 885.538,A 0.000,B 0.000,C 90.000,E1 132.771} C_DIS
LIN {X -0.091,Y -627.452,Z 885.530,A 0.000,B 0.000,C 90.000,E1 131.472} C_DIS
LIN {X -0.008,Y -630.646,Z 885.526,A 0.000,B 0.000,C 90.000,E1 130.701} C_DIS
LIN {X -0.050,Y -635.723,Z 885.519,A 0.000,B 0.000,C 90.000,E1 129.439} C_DIS
LIN {X -0.115,Y -641.654,Z 885.511,A 0.000,B 0.000,C 90.000,E1 127.935} C_DIS
LIN {X 0.134,Y -646.532,Z 885.504,A 0.000,B 0.000,C 90.000,E1 126.664} C_DIS
LIN {X -0.055,Y -650.990,Z 885.497,A 0.000,B 0.000,C 90.000,E1 125.438} C_DIS
LIN {X -0.019,Y -655.194,Z 885.490,A 0.000,B 0.000,C 90.000,E1 124.199} C_DIS
LIN {X -0.013,Y -658.283,Z 885.485,A 0.000,B 0.000,C 90.000,E1 123.214} C_DIS
LIN {X -0.357,Y -659.810,Z 885.482,A 0.000,B 0.000,C 90.000,E1 122.752} C_DIS
LIN {X -0.094,Y -662.367,Z 885.476,A 0.000,B 0.000,C 90.000,E1 121.750} C_DIS
LIN {X 0.074,Y -664.052,Z 885.472,A 0.000,B 0.000,C 90.000,E1 121.003} C_DIS
LIN {X -0.181,Y -665.936,Z 885.467,A 0.000,B 0.000,C 90.000,E1 120.050} C_DIS
LIN {X -0.170,Y -667.592,Z 885.461,A 0.000,B 0.000,C 90.000,E1 119.077} C_DIS
LIN {X -0.290,Y -668.742,Z 885.457,A 0.000,B 0.000,C 90.000,E1 118.359} C_DIS
LIN {X 0.092,Y -670.894,Z 885.449,A 0.000,B 0.000,C 90.000,E1 116.873} C_DIS
LIN {X 0.044,Y -672.082,Z 885.443,A 0.000,B 0.000,C 90.000,E1 115.668} C_DIS
LIN {X -0.047,Y -672.549,Z 885.439,A 0.000,B 0.000,C 90.000,E1 114.951} C_DIS
LIN {X 0.191,Y -672.811,Z 885.435,A 0.000,B 0.000,C 90.000,E1 114.207} C_DIS
LIN {X -0.352,Y -672.651,Z 885.432,A 0.000,B 0.000,C 90.000,E1 113.770} C_DIS
LIN {X -0.180,Y -672.510,Z 885.431,A 0.000,B 0.000,C 90.000,E1 113.515} C_DIS
LIN {X -0.106,Y -671.603,Z 885.428,A 0.000,B 0.000,C 90.000,E1 113.025} C_DIS
LIN {X 0.062,Y -670.861,Z 885.427,A 0.000,B 0.000,C 90.000,E1 112.770} C_DIS
LIN {X 0.128,Y -667.994,Z 885.424,A 0.000,B 0.000,C 90.000,E1 112.280} C_DIS
LIN {X 0.204,Y -667.114,Z 885.423,A 0.000,B 0.000,C 90.000,E1 112.153} C_DIS
LIN {X 0.280,Y -665.735,Z 885.423,A 0.000,B 0.000,C 90.000,E1 112.025} C_DIS
LIN {X -0.252,Y -662.526,Z 885.421,A 0.000,B 0.000,C 90.000,E1 111.844} C_DIS
LIN {X 0.376,Y -660.203,Z 885.420,A 0.000,B 0.000,C 90.000,E1 111.589} C_DIS
LIN {X -0.310,Y -657.888,Z 885.420,A 0.000,B 0.000,C 90.000,E1 111.535} C_DIS
LIN {X -0.036,Y -651.997,Z 885.418,A 0.000,B 0.000,C 90.000,E1 111.280} C_DIS
LIN {X -0.116,Y -647.439,Z 885.417,A 0.000,B 0.000,C 90.000,E1 111.153} C_DIS
LIN {X -0.078,Y -631.052,Z 885.415,A 0.000,B 0.000,C 90.000,E1 110.737} C_DIS
LIN {X -0.119,Y -619.370,Z 885.413,A 0.000,B 0.000,C 90.000,E1 110.429} C_DIS
LIN {X -0.184,Y -610.308,Z 885.412,A 0.000,B 0.000,C 90.000,E1 110.120} C_DIS
LIN {X -0.015,Y -604.669,Z 885.410,A 0.000,B 0.000,C 90.000,E1 109.866} C_DIS
LIN {X -0.258,Y -595.616,Z 885.408,A 0.000,B 0.000,C 90.000,E1 109.450} C_DIS
LIN {X -0.132,Y -587.799,Z 885.406,A 0.000,B 0.000,C 90.000,E1 109.033} C_DIS
LIN {X 0.294,Y -579.129,Z 885.404,A 0.000,B 0.000,C 90.000,E1 108.598} C_DIS
LIN {X 0.063,Y -567.847,Z 885.401,A 0.000,B 0.000,C 90.000,E1 108.236} C_DIS
LIN {X 0.005,Y -564.423,Z 885.401,A 0.000,B 0.000,C 90.000,E1 108.127} C_DIS
LIN {X -0.123,Y -562.446,Z 885.400,A 0.000,B 0.000,C 90.000,E1 108.055} C_DIS
LIN {X 0.029,Y -558.943,Z 885.399,A 0.000,B 0.000,C 90.000,E1 107.819} C_DIS
LIN {X -0.002,Y -558.924,Z 885.399,A 0.000,B 0.000,C 90.000,E1 107.819} C_DIS
LIN {X 0.041,Y -557.609,Z 885.398,A 0.000,B 0.000,C 90.000,E1 107.583} C_DIS
LIN {X -0.149,Y -556.954,Z 885.396,A 0.000,B 0.000,C 90.000,E1 107.221} C_DIS
LIN {X 0.181,Y -556.862,Z 885.391,A 0.000,B 0.000,C 90.000,E1 106.441} C_DIS
LIN {X 0.319,Y -557.803,Z 885.376,A 0.000,B 0.000,C 90.000,E1 103.647} C_DIS
LIN {X -0.190,Y -559.092,Z 885.364,A 0.000,B 0.000,C 90.000,E1 101.478} C_DIS
LIN {X 0.186,Y -560.514,Z 885.353,A 0.000,B 0.000,C 90.000,E1 99.500} C_DIS
LIN {X -0.265,Y -561.433,Z 885.345,A 0.000,B 0.000,C 90.000,E1 98.163} C_DIS
LIN {X -0.227,Y -562.316,Z 885.338,A 0.000,B 0.000,C 90.000,E1 96.777} C_DIS
LIN {X 0.238,Y -562.956,Z 885.331,A 0.000,B 0.000,C 90.000,E1 95.625} C_DIS
LIN {X -0.175,Y -563.710,Z 885.322,A 0.000,B 0.000,C 90.000,E1 94.012} C_DIS
LIN {X -0.196,Y -564.214,Z 885.315,A 0.000,B 0.000,C 90.000,E1 92.636} C_DIS
LIN {X -0.096,Y -564.742,Z 885.305,A 0.000,B 0.000,C 90.000,E1 90.974} C_DIS
LIN {X -0.107,Y -565.088,Z 885.298,A 0.000,B 0.000,C 90.000,E1 89.599} C_DIS
LIN {X -0.116,Y -565.426,Z 885.290,A 0.000,B 0.000,C 90.000,E1 88.224} C_DIS
LIN {X 0.031,Y -565.677,Z 885.281,A 0.000,B 0.000,C 90.000,E1 86.560} C_DIS
LIN {X 0.088,Y -565.917,Z 885.273,A 0.000,B 0.000,C 90.000,E1 85.179} C_DIS
LIN {X -0.153,Y -566.243,Z 885.263,A 0.000,B 0.000,C 90.000,E1 83.280} C_DIS
LIN {X -0.164,Y -566.794,Z 885.250,A 0.000,B 0.000,C 90.000,E1 81.084} C_DIS
LIN {X -0.157,Y -567.497,Z 885.240,A 0.000,B 0.000,C 90.000,E1 79.162} C_DIS
LIN {X -0.017,Y -568.397,Z 885.229,A 0.000,B 0.000,C 90.000,E1 77.229} C_DIS
LIN {X -0.227,Y -568.982,Z 885.221,A 0.000,B 0.000,C 90.000,E1 75.880} C_DIS
LIN {X 0.077,Y -569.470,Z 885.215,A 0.000,B 0.000,C 90.000,E1 74.755} C_DIS
LIN {X -0.162,Y -569.895,Z 885.209,A 0.000,B 0.000,C 90.000,E1 73.685} C_DIS
LIN {X -0.093,Y -570.383,Z 885.199,A 0.000,B 0.000,C 90.000,E1 71.764} C_DIS
LIN {X 0.164,Y -570.735,Z 885.188,A 0.000,B 0.000,C 90.000,E1 69.826} C_DIS
LIN {X 0.087,Y -570.893,Z 885.177,A 0.000,B 0.000,C 90.000,E1 67.922} C_DIS
LIN {X 0.048,Y -571.035,Z 885.170,A 0.000,B 0.000,C 90.000,E1 66.561} C_DIS
LIN {X -0.102,Y -571.012,Z 885.159,A 0.000,B 0.000,C 90.000,E1 64.665} C_DIS
LIN {X -0.174,Y -570.933,Z 885.152,A 0.000,B 0.000,C 90.000,E1 63.307} C_DIS
LIN {X 0.098,Y -570.605,Z 885.143,A 0.000,B 0.000,C 90.000,E1 61.641} C_DIS
LIN {X 0.015,Y -570.306,Z 885.135,A 0.000,B 0.000,C 90.000,E1 60.284} C_DIS
LIN {X -0.050,Y -570.150,Z 885.132,A 0.000,B 0.000,C 90.000,E1 59.744} C_DIS
LIN {X 0.361,Y -569.071,Z 885.121,A 0.000,B 0.000,C 90.000,E1 57.788} C_DIS
LIN {X 0.103,Y -568.506,Z 885.117,A 0.000,B 0.000,C 90.000,E1 56.993} C_DIS
LIN {X -0.086,Y -567.321,Z 885.109,A 0.000,B 0.000,C 90.000,E1 55.642} C_DIS
LIN {X -0.050,Y -566.492,Z 885.105,A 0.000,B 0.000,C 90.000,E1 54.815} C_DIS
LIN {X -0.029,Y -565.512,Z 885.100,A 0.000,B 0.000,C 90.000,E1 53.989} C_DIS
LIN {X 0.311,Y -564.389,Z 885.095,A 0.000,B 0.000,C 90.000,E1 53.130} C_DIS
LIN {X -0.048,Y -562.739,Z 885.089,A 0.000,B 0.000,C 90.000,E1 52.065} C_DIS
LIN {X -0.184,Y -561.338,Z 885.085,A 0.000,B 0.000,C 90.000,E1 51.251} C_DIS
LIN {X -0.331,Y -559.711,Z 885.080,A 0.000,B 0.000,C 90.000,E1 50.436} C_DIS
LIN {X -0.135,Y -557.887,Z 885.075,A 0.000,B 0.000,C 90.000,E1 49.585} C_DIS
LIN {X 0.027,Y -556.497,Z 885.072,A 0.000,B 0.000,C 90.000,E1 49.013} C_DIS
LIN {X 0.122,Y -554.956,Z 885.069,A 0.000,B 0.000,C 90.000,E1 48.447} C_DIS
LIN {X -0.099,Y -552.350,Z 885.065,A 0.000,B 0.000,C 90.000,E1 47.634} C_DIS
LIN {X 0.019,Y -549.422,Z 885.060,A 0.000,B 0.000,C 90.000,E1 46.782} C_DIS
LIN {X -0.293,Y -546.275,Z 885.055,A 0.000,B 0.000,C 90.000,E1 45.972} C_DIS
LIN {X 0.112,Y -545.203,Z 885.054,A 0.000,B 0.000,C 90.000,E1 45.648} C_DIS
LIN {X -0.050,Y -542.208,Z 885.050,A 0.000,B 0.000,C 90.000,E1 44.960} C_DIS
LIN {X -0.240,Y -538.810,Z 885.046,A 0.000,B 0.000,C 90.000,E1 44.271} C_DIS
LIN {X -0.264,Y -535.866,Z 885.043,A 0.000,B 0.000,C 90.000,E1 43.704} C_DIS
LIN {X 0.250,Y -531.791,Z 885.039,A 0.000,B 0.000,C 90.000,E1 42.933} C_DIS
LIN {X 0.170,Y -528.326,Z 885.036,A 0.000,B 0.000,C 90.000,E1 42.366} C_DIS
LIN {X -0.287,Y -524.672,Z 885.032,A 0.000,B 0.000,C 90.000,E1 41.838} C_DIS
LIN {X -0.176,Y -521.859,Z 885.030,A 0.000,B 0.000,C 90.000,E1 41.391} C_DIS
LIN {X 0.134,Y -514.490,Z 885.024,A 0.000,B 0.000,C 90.000,E1 40.334} C_DIS
LIN {X -0.285,Y -508.799,Z 885.020,A 0.000,B 0.000,C 90.000,E1 39.644} C_DIS
LIN {X -0.047,Y -502.578,Z 885.016,A 0.000,B 0.000,C 90.000,E1 38.874} C_DIS
LIN {X 0.157,Y -497.270,Z 885.013,A 0.000,B 0.000,C 90.000,E1 38.257} C_DIS
LIN {X -0.069,Y -490.346,Z 885.009,A 0.000,B 0.000,C 90.000,E1 37.569} C_DIS
LIN {X -0.047,Y -483.273,Z 885.005,A 0.000,B 0.000,C 90.000,E1 36.870} C_DIS
LIN {X -0.202,Y -475.911,Z 885.001,A 0.000,B 0.000,C 90.000,E1 36.217} C_DIS
LIN {X -0.227,Y -465.310,Z 884.996,A 0.000,B 0.000,C 90.000,E1 35.311} C_DIS
LIN {X -0.166,Y -453.428,Z 884.991,A 0.000,B 0.000,C 90.000,E1 34.326} C_DIS
LIN {X -0.217,Y -436.294,Z 884.983,A 0.000,B 0.000,C 90.000,E1 32.959} C_DIS
LIN {X -0.071,Y -416.478,Z 884.974,A 0.000,B 0.000,C 90.000,E1 31.258} C_DIS
LIN {X -0.017,Y -403.182,Z 884.967,A 0.000,B 0.000,C 90.000,E1 30.001} C_DIS
LIN {X -0.159,Y -397.476,Z 884.963,A 0.000,B 0.000,C 90.000,E1 29.411} C_DIS
LIN {X 0.165,Y -395.117,Z 884.962,A 0.000,B 0.000,C 90.000,E1 29.077} C_DIS
LIN {X 0.072,Y -394.162,Z 884.961,A 0.000,B 0.000,C 90.000,E1 28.949} C_DIS
LIN {X 0.178,Y -392.605,Z 884.959,A 0.000,B 0.000,C 90.000,E1 28.615} C_DIS
LIN {X -0.157,Y -391.581,Z 884.958,A 0.000,B 0.000,C 90.000,E1 28.487} C_DIS
LIN {X 0.036,Y -390.980,Z 884.957,A 0.000,B 0.000,C 90.000,E1 28.281} C_DIS
LIN {X -0.028,Y -389.770,Z 884.955,A 0.000,B 0.000,C 90.000,E1 27.847} C_DIS
LIN {X 0.082,Y -389.297,Z 884.952,A 0.000,B 0.000,C 90.000,E1 27.385} C_DIS
LIN {X -0.076,Y -389.087,Z 884.950,A 0.000,B 0.000,C 90.000,E1 27.052} C_DIS
LIN {X 0.000,Y -389.273,Z 884.944,A 0.000,B 0.000,C 90.000,E1 25.976} C_DIS
LIN {X -0.138,Y -392.261,Z 884.923,A 0.000,B 0.000,C 90.000,E1 22.078} C_DIS
LIN {X 0.054,Y -395.189,Z 884.907,A 0.000,B 0.000,C 90.000,E1 19.214} C_DIS
LIN {X 0.144,Y -398.055,Z 884.893,A 0.000,B 0.000,C 90.000,E1 16.732} C_DIS
LIN {X -0.033,Y -401.204,Z 884.879,A 0.000,B 0.000,C 90.000,E1 14.300} C_DIS
LIN {X 0.179,Y -405.563,Z 884.862,A 0.000,B 0.000,C 90.000,E1 11.130} C_DIS
LIN {X -0.095,Y -408.244,Z 884.852,A 0.000,B 0.000,C 90.000,E1 9.434} C_DIS
LIN {X -0.010,Y -412.868,Z 884.837,A 0.000,B 0.000,C 90.000,E1 6.663} C_DIS
LIN {X 0.189,Y -418.021,Z 884.822,A 0.000,B 0.000,C 90.000,E1 3.898} C_DIS
LIN {X 0.139,Y -425.202,Z 884.803,A 0.000,B 0.000,C 90.000,E1 0.516} C_DIS
LIN {X 0.072,Y -430.999,Z 884.790,A 0.000,B 0.000,C 90.000,E1 358.108} C_DIS
LIN {X -0.165,Y -437.113,Z 884.777,A 0.000,B 0.000,C 90.000,E1 355.812} C_DIS
LIN {X -0.024,Y -438.757,Z 884.774,A 0.000,B 0.000,C 90.000,E1 355.298} C_DIS
LIN {X 0.060,Y -439.443,Z 884.773,A 0.000,B 0.000,C 90.000,E1 355.122} C_DIS
LIN {X 0.153,Y -441.500,Z 884.771,A 0.000,B 0.000,C 90.000,E1 354.723} C_DIS
LIN {X -0.207,Y -443.921,Z 884.769,A 0.000,B 0.000,C 90.000,E1 354.432} C_DIS
LIN {X -0.094,Y -447.962,Z 884.767,A 0.000,B 0.000,C 90.000,E1 354.090} C_DIS
LIN {X 0.027,Y -449.512,Z 884.767,A 0.000,B 0.000,C 90.000,E1 353.970} C_DIS
LIN {X 0.157,Y -454.948,Z 884.765,A 0.000,B 0.000,C 90.000,E1 353.685} C_DIS
LIN {X -0.171,Y -469.053,Z 884.762,A 0.000,B 0.000,C 90.000,E1 353.109} C_DIS
LIN {X 0.061,Y -475.679,Z 884.760,A 0.000,B 0.000,C 90.000,E1 352.761} C_DIS
LIN {X 0.120,Y -482.328,Z 884.758,A 0.000,B 0.000,C 90.000,E1 352.413} C_DIS
LIN {X -0.140,Y -492.226,Z 884.755,A 0.000,B 0.000,C 90.000,E1 351.894} C_DIS
LIN {X -0.113,Y -502.055,Z 884.752,A 0.000,B 0.000,C 90.000,E1 351.319} C_DIS
LIN {X -0.246,Y -511.513,Z 884.748,A 0.000,B 0.000,C 90.000,E1 350.735} C_DIS
LIN {X -0.032,Y -519.145,Z 884.746,A 0.000,B 0.000,C 90.000,E1 350.208} C_DIS
LIN {X -0.120,Y -528.282,Z 884.742,A 0.000,B 0.000,C 90.000,E1 349.567} C_DIS
LIN {X -0.034,Y -534.167,Z 884.740,A 0.000,B 0.000,C 90.000,E1 349.106} C_DIS
LIN {X -0.010,Y -539.958,Z 884.737,A 0.000,B 0.000,C 90.000,E1 348.634} C_DIS
LIN {X 0.107,Y -548.237,Z 884.733,A 0.000,B 0.000,C 90.000,E1 347.881} C_DIS
LIN {X 0.220,Y -554.904,Z 884.729,A 0.000,B 0.000,C 90.000,E1 347.229} C_DIS
LIN {X -0.278,Y -560.983,Z 884.726,A 0.000,B 0.000,C 90.000,E1 346.645} C_DIS
LIN {X -0.150,Y -568.249,Z 884.721,A 0.000,B 0.000,C 90.000,E1 345.811} C_DIS
LIN {X 0.093,Y -573.850,Z 884.717,A 0.000,B 0.000,C 90.000,E1 345.102} C_DIS
LIN {X 0.136,Y -580.107,Z 884.713,A 0.000,B 0.000,C 90.000,E1 344.283} C_DIS
LIN {X 0.085,Y -584.936,Z 884.709,A 0.000,B 0.000,C 90.000,E1 343.614} C_DIS
LIN {X -0.161,Y -590.336,Z 884.705,A 0.000,B 0.000,C 90.000,E1 342.834} C_DIS
LIN {X -0.096,Y -596.922,Z 884.699,A 0.000,B 0.000,C 90.000,E1 341.764} C_DIS
LIN {X 0.240,Y -602.932,Z 884.693,A 0.000,B 0.000,C 90.000,E1 340.678} C_DIS
LIN {X -0.203,Y -607.194,Z 884.688,A 0.000,B 0.000,C 90.000,E1 339.934} C_DIS
LIN {X 0.249,Y -613.201,Z 884.682,A 0.000,B 0.000,C 90.000,E1 338.720} C_DIS
LIN {X -0.101,Y -617.690,Z 884.677,A 0.000,B 0.000,C 90.000,E1 337.847} C_DIS
LIN {X 0.173,Y -621.898,Z 884.672,A 0.000,B 0.000,C 90.000,E1 336.922} C_DIS
LIN {X -0.081,Y -626.453,Z 884.666,A 0.000,B 0.000,C 90.000,E1 335.921} C_DIS
LIN {X -0.281,Y -630.697,Z 884.661,A 0.000,B 0.000,C 90.000,E1 334.921} C_DIS
LIN {X -0.157,Y -634.654,Z 884.655,A 0.000,B 0.000,C 90.000,E1 333.896} C_DIS
LIN {X 0.025,Y -638.327,Z 884.649,A 0.000,B 0.000,C 90.000,E1 332.871} C_DIS
LIN {X 0.134,Y -640.076,Z 884.647,A 0.000,B 0.000,C 90.000,E1 332.359} C_DIS
LIN {X -0.183,Y -643.385,Z 884.641,A 0.000,B 0.000,C 90.000,E1 331.385} C_DIS
LIN {X -0.142,Y -646.386,Z 884.635,A 0.000,B 0.000,C 90.000,E1 330.383} C_DIS
LIN {X -0.383,Y -649.352,Z 884.630,A 0.000,B 0.000,C 90.000,E1 329.410} C_DIS
LIN {X 0.169,Y -652.811,Z 884.623,A 0.000,B 0.000,C 90.000,E1 328.122} C_DIS
LIN {X 0.243,Y -654.696,Z 884.619,A 0.000,B 0.000,C 90.000,E1 327.375} C_DIS
LIN {X -0.021,Y -657.462,Z 884.612,A 0.000,B 0.000,C 90.000,E1 326.167} C_DIS
LIN {X 0.016,Y -659.451,Z 884.607,A 0.000,B 0.000,C 90.000,E1 325.182} C_DIS
LIN {X -0.358,Y -661.459,Z 884.600,A 0.000,B 0.000,C 90.000,E1 323.989} C_DIS
LIN {X 0.171,Y -662.546,Z 884.596,A 0.000,B 0.000,C 90.000,E1 323.210} C_DIS
LIN {X -0.256,Y -663.844,Z 884.590,A 0.000,B 0.000,C 90.000,E1 322.271} C_DIS
LIN {X 0.245,Y -665.195,Z 884.584,A 0.000,B 0.000,C 90.000,E1 321.009} C_DIS
LIN {X 0.333,Y -666.695,Z 884.575,A 0.000,B 0.000,C 90.000,E1 319.542} C_DIS
LIN {X -0.122,Y -667.476,Z 884.571,A 0.000,B 0.000,C 90.000,E1 318.852} C_DIS
LIN {X -0.060,Y -669.327,Z 884.562,A 0.000,B 0.000,C 90.000,E1 317.148} C_DIS
LIN {X 0.020,Y -670.860,Z 884.554,A 0.000,B 0.000,C 90.000,E1 315.688} C_DIS
LIN {X -0.382,Y -672.098,Z 884.547,A 0.000,B 0.000,C 90.000,E1 314.514} C_DIS
LIN {X 0.244,Y -673.773,Z 884.538,A 0.000,B 0.000,C 90.000,E1 312.771} C_DIS
LIN {X -0.100,Y -674.954,Z 884.531,A 0.000,B 0.000,C 90.000,E1 311.595} C_DIS
LIN {X -0.344,Y -676.163,Z 884.523,A 0.000,B 0.000,C 90.000,E1 310.172} C_DIS
LIN {X -0.157,Y -677.200,Z 884.516,A 0.000,B 0.000,C 90.000,E1 308.955} C_DIS
LIN {X -0.256,Y -678.312,Z 884.508,A 0.000,B 0.000,C 90.000,E1 307.523} C_DIS
LIN {X 0.071,Y -679.205,Z 884.502,A 0.000,B 0.000,C 90.000,E1 306.297} C_DIS
LIN {X 0.009,Y -679.989,Z 884.495,A 0.000,B 0.000,C 90.000,E1 305.105} C_DIS
LIN {X 0.127,Y -680.951,Z 884.486,A 0.000,B 0.000,C 90.000,E1 303.420} C_DIS
LIN {X 0.282,Y -681.773,Z 884.479,A 0.000,B 0.000,C 90.000,E1 302.212} C_DIS
LIN {X -0.311,Y -683.074,Z 884.470,A 0.000,B 0.000,C 90.000,E1 300.590} C_DIS
LIN {X -0.207,Y -684.997,Z 884.458,A 0.000,B 0.000,C 90.000,E1 298.437} C_DIS
LIN {X 0.120,Y -686.837,Z 884.449,A 0.000,B 0.000,C 90.000,E1 296.744} C_DIS
LIN {X -0.061,Y -688.557,Z 884.441,A 0.000,B 0.000,C 90.000,E1 295.335} C_DIS
LIN {X 0.171,Y -689.698,Z 884.434,A 0.000,B 0.000,C 90.000,E1 294.131} C_DIS
LIN {X -0.049,Y -690.190,Z 884.430,A 0.000,B 0.000,C 90.000,E1 293.439} C_DIS
LIN {X 0.140,Y -689.952,Z 884.428,A 0.000,B 0.000,C 90.000,E1 292.950} C_DIS
LIN {X 0.102,Y -689.686,Z 884.426,A 0.000,B 0.000,C 90.000,E1 292.717} C_DIS
LIN {X -0.081,Y -688.210,Z 884.424,A 0.000,B 0.000,C 90.000,E1 292.259} C_DIS
LIN {X -0.118,Y -687.189,Z 884.422,A 0.000,B 0.000,C 90.000,E1 292.025} C_DIS
LIN {X -0.008,Y -686.273,Z 884.422,A 0.000,B 0.000,C 90.000,E1 291.897} C_DIS
LIN {X 0.356,Y -681.112,Z 884.419,A 0.000,B 0.000,C 90.000,E1 291.408} C_DIS
LIN {X -0.090,Y -679.509,Z 884.419,A 0.000,B 0.000,C 90.000,E1 291.334} C_DIS
LIN {X 0.002,Y -677.173,Z 884.418,A 0.000,B 0.000,C 90.000,E1 291.227} C_DIS
LIN {X -0.042,Y -668.890,Z 884.417,A 0.000,B 0.000,C 90.000,E1 290.972} C_DIS
LIN {X -0.220,Y -661.764,Z 884.415,A 0.000,B 0.000,C 90.000,E1 290.791} C_DIS
LIN {X -0.138,Y -659.014,Z 884.415,A 0.000,B 0.000,C 90.000,E1 290.663} C_DIS
LIN {X -0.106,Y -656.382,Z 884.414,A 0.000,B 0.000,C 90.000,E1 290.536} C_DIS
LIN {X -0.162,Y -656.320,Z 884.414,A 0.000,B 0.000,C 90.000,E1 290.536} C_DIS
LIN {X 0.176,Y -655.212,Z 884.413,A 0.000,B 0.000,C 90.000,E1 290.375} C_DIS
LIN {X 0.131,Y -655.181,Z 884.413,A 0.000,B 0.000,C 90.000,E1 290.375} C_DIS
LIN {X 0.051,Y -655.088,Z 884.413,A 0.000,B 0.000,C 90.000,E1 290.248} C_DIS
LIN {X 0.099,Y -655.219,Z 884.412,A 0.000,B 0.000,C 90.000,E1 290.120} C_DIS
LIN {X 0.018,Y -656.272,Z 884.410,A 0.000,B 0.000,C 90.000,E1 289.758} C_DIS
LIN {X -0.128,Y -659.795,Z 884.406,A 0.000,B 0.000,C 90.000,E1 289.033} C_DIS
LIN {X -0.126,Y -665.028,Z 884.400,A 0.000,B 0.000,C 90.000,E1 288.055} C_DIS
LIN {X -0.219,Y -666.308,Z 884.399,A 0.000,B 0.000,C 90.000,E1 287.819} C_DIS
LIN {X -0.273,Y -669.687,Z 884.395,A 0.000,B 0.000,C 90.000,E1 287.094} C_DIS
LIN {X 0.221,Y -671.700,Z 884.392,A 0.000,B 0.000,C 90.000,E1 286.567} C_DIS
LIN {X 0.217,Y -674.227,Z 884.388,A 0.000,B 0.000,C 90.000,E1 285.843} C_DIS
LIN {X 0.050,Y -676.129,Z 884.384,A 0.000,B 0.000,C 90.000,E1 285.134} C_DIS
LIN {X 0.075,Y -677.685,Z 884.380,A 0.000,B 0.000,C 90.000,E1 284.411} C_DIS
LIN {X -0.061,Y -678.943,Z 884.376,A 0.000,B 0.000,C 90.000,E1 283.703} C_DIS
LIN {X -0.340,Y -679.985,Z 884.372,A 0.000,B 0.000,C 90.000,E1 283.008} C_DIS
LIN {X 0.215,Y -680.676,Z 884.368,A 0.000,B 0.000,C 90.000,E1 282.243} C_DIS
LIN {X 0.105,Y -681.075,Z 884.364,A 0.000,B 0.000,C 90.000,E1 281.535} C_DIS
LIN {X 0.068,Y -681.156,Z 884.363,A 0.000,B 0.000,C 90.000,E1 281.299} C_DIS
LIN {X -0.175,Y -680.758,Z 884.359,A 0.000,B 0.000,C 90.000,E1 280.602} C_DIS
LIN {X -0.376,Y -680.270,Z 884.356,A 0.000,B 0.000,C 90.000,E1 280.141} C_DIS
LIN {X 0.210,Y -679.498,Z 884.354,A 0.000,B 0.000,C 90.000,E1 279.613} C_DIS
LIN {X 0.006,Y -678.362,Z 884.351,A 0.000,B 0.000,C 90.000,E1 279.151} C_DIS
LIN {X -0.257,Y -676.106,Z 884.347,A 0.000,B 0.000,C 90.000,E1 278.454} C_DIS
LIN {X 0.193,Y -674.288,Z 884.344,A 0.000,B 0.000,C 90.000,E1 277.936} C_DIS
LIN {X 0.053,Y -672.160,Z 884.342,A 0.000,B 0.000,C 90.000,E1 277.466} C_DIS
LIN {X -0.276,Y -669.078,Z 884.338,A 0.000,B 0.000,C 90.000,E1 276.891} C_DIS
LIN {X 0.036,Y -665.565,Z 884.335,A 0.000,B 0.000,C 90.000,E1 276.258} C_DIS
LIN {X -0.251,Y -662.407,Z 884.332,A 0.000,B 0.000,C 90.000,E1 275.796} C_DIS
LIN {X 0.099,Y -658.794,Z 884.329,A 0.000,B 0.000,C 90.000,E1 275.277} C_DIS
LIN {X -0.289,Y -654.714,Z 884.327,A 0.000,B 0.000,C 90.000,E1 274.821} C_DIS
LIN {X -0.096,Y -648.856,Z 884.323,A 0.000,B 0.000,C 90.000,E1 274.188} C_DIS
LIN {X 0.258,Y -643.801,Z 884.321,A 0.000,B 0.000,C 90.000,E1 273.669} C_DIS
LIN {X 0.205,Y -637.149,Z 884.317,A 0.000,B 0.000,C 90.000,E1 273.094} C_DIS
LIN {X -0.282,Y -631.615,Z 884.315,A 0.000,B 0.000,C 90.000,E1 272.694} C_DIS
LIN {X 0.214,Y -624.061,Z 884.312,A 0.000,B 0.000,C 90.000,E1 272.121} C_DIS
LIN {X -0.190,Y -617.798,Z 884.310,A 0.000,B 0.000,C 90.000,E1 271.776} C_DIS
LIN {X 0.302,Y -611.325,Z 884.308,A 0.000,B 0.000,C 90.000,E1 271.375} C_DIS
LIN {X -0.104,Y -604.543,Z 884.306,A 0.000,B 0.000,C 90.000,E1 271.088} C_DIS
LIN {X -0.216,Y -597.660,Z 884.304,A 0.000,B 0.000,C 90.000,E1 270.802} C_DIS
LIN {X 0.045,Y -590.445,Z 884.303,A 0.000,B 0.000,C 90.000,E1 270.516} C_DIS
LIN {X 0.166,Y -583.107,Z 884.302,A 0.000,B 0.000,C 90.000,E1 270.286} C_DIS
LIN {X -0.113,Y -577.728,Z 884.301,A 0.000,B 0.000,C 90.000,E1 270.172} C_DIS
LIN {X -0.268,Y -571.230,Z 884.300,A 0.000,B 0.000,C 90.000,E1 270.057} C_DIS
LIN {X 0.018,Y -564.146,Z 884.300,A 0.000,B 0.000,C 90.000,E1 269.943} C_DIS
LIN {X -0.205,Y -552.576,Z 884.299,A 0.000,B 0.000,C 90.000,E1 269.885} C_DIS
LIN {X 0.215,Y -549.809,Z 884.299,A 0.000,B 0.000,C 90.000,E1 269.771} C_DIS
LIN {X 0.166,Y -549.652,Z 884.299,A 0.000,B 0.000,C 90.000,E1 269.771} C_DIS
LIN {X -0.076,Y -546.358,Z 884.297,A 0.000,B 0.000,C 90.000,E1 269.427} C_DIS
LIN {X -0.117,Y -546.320,Z 884.297,A 0.000,B 0.000,C 90.000,E1 269.427} C_DIS
LIN {X 0.223,Y -545.218,Z 884.294,A 0.000,B 0.000,C 90.000,E1 268.912} C_DIS
LIN {X -0.080,Y -543.498,Z 884.286,A 0.000,B 0.000,C 90.000,E1 267.535} C_DIS
LIN {X -0.279,Y -541.370,Z 884.271,A 0.000,B 0.000,C 90.000,E1 264.723} C_DIS
LIN {X -0.065,Y -540.446,Z 884.263,A 0.000,B 0.000,C 90.000,E1 263.280} C_DIS
LIN {X 0.066,Y -539.534,Z 884.256,A 0.000,B 0.000,C 90.000,E1 262.129} C_DIS
LIN {X -0.215,Y -538.154,Z 884.248,A 0.000,B 0.000,C 90.000,E1 260.735} C_DIS
LIN {X 0.129,Y -536.069,Z 884.237,A 0.000,B 0.000,C 90.000,E1 258.701} C_DIS
LIN {X 0.003,Y -534.538,Z 884.229,A 0.000,B 0.000,C 90.000,E1 257.285} C_DIS
LIN {X -0.267,Y -532.760,Z 884.221,A 0.000,B 0.000,C 90.000,E1 255.880} C_DIS
LIN {X 0.235,Y -530.583,Z 884.212,A 0.000,B 0.000,C 90.000,E1 254.102} C_DIS
LIN {X -0.164,Y -528.176,Z 884.201,A 0.000,B 0.000,C 90.000,E1 252.127} C_DIS
LIN {X 0.193,Y -527.078,Z 884.196,A 0.000,B 0.000,C 90.000,E1 251.221} C_DIS
LIN {X -0.127,Y -524.848,Z 884.186,A 0.000,B 0.000,C 90.000,E1 249.518} C_DIS
LIN {X 0.048,Y -523.311,Z 884.180,A 0.000,B 0.000,C 90.000,E1 248.337} C_DIS
LIN {X 0.160,Y -521.176,Z 884.172,A 0.000,B 0.000,C 90.000,E1 246.869} C_DIS
LIN {X -0.198,Y -519.399,Z 884.165,A 0.000,B 0.000,C 90.000,E1 245.741} C_DIS
LIN {X -0.225,Y -517.189,Z 884.157,A 0.000,B 0.000,C 90.000,E1 244.280} C_DIS
LIN {X -0.075,Y -515.788,Z 884.152,A 0.000,B 0.000,C 90.000,E1 243.384} C_DIS
LIN {X -0.281,Y -512.713,Z 884.142,A 0.000,B 0.000,C 90.000,E1 241.641} C_DIS
LIN {X -0.314,Y -509.641,Z 884.132,A 0.000,B 0.000,C 90.000,E1 239.871} C_DIS
LIN {X -0.117,Y -507.579,Z 884.126,A 0.000,B 0.000,C 90.000,E1 238.663} C_DIS
LIN {X -0.060,Y -504.808,Z 884.118,A 0.000,B 0.000,C 90.000,E1 237.168} C_DIS
LIN {X -0.060,Y -501.772,Z 884.109,A 0.000,B 0.000,C 90.000,E1 235.674} C_DIS
LIN {X 0.117,Y -500.431,Z 884.106,A 0.000,B 0.000,C 90.000,E1 235.055} C_DIS
LIN {X -0.106,Y -496.894,Z 884.098,A 0.000,B 0.000,C 90.000,E1 233.577} C_DIS
LIN {X 0.185,Y -494.882,Z 884.093,A 0.000,B 0.000,C 90.000,E1 232.637} C_DIS
LIN {X -0.072,Y -490.674,Z 884.083,A 0.000,B 0.000,C 90.000,E1 230.848} C_DIS
LIN {X -0.040,Y -486.482,Z 884.072,A 0.000,B 0.000,C 90.000,E1 229.013} C_DIS
LIN {X 0.071,Y -484.417,Z 884.067,A 0.000,B 0.000,C 90.000,E1 228.081} C_DIS
LIN {X 0.224,Y -480.382,Z 884.057,A 0.000,B 0.000,C 90.000,E1 226.215} C_DIS
LIN {X -0.202,Y -478.972,Z 884.054,A 0.000,B 0.000,C 90.000,E1 225.648} C_DIS
LIN {X -0.295,Y -475.531,Z 884.045,A 0.000,B 0.000,C 90.000,E1 224.109} C_DIS
LIN {X -0.250,Y -470.625,Z 884.033,A 0.000,B 0.000,C 90.000,E1 221.919} C_DIS
LIN {X 0.000,Y -465.798,Z 884.021,A 0.000,B 0.000,C 90.000,E1 219.688} C_DIS
LIN {X -0.163,Y -461.738,Z 884.010,A 0.000,B 0.000,C 90.000,E1 217.810} C_DIS
LIN {X -0.040,Y -457.721,Z 883.999,A 0.000,B 0.000,C 90.000,E1 215.884} C_DIS
LIN {X -0.275,Y -453.663,Z 883.989,A 0.000,B 0.000,C 90.000,E1 213.992} C_DIS
LIN {X -0.031,Y -450.844,Z 883.982,A 0.000,B 0.000,C 90.000,E1 212.673} C_DIS
LIN {X -0.080,Y -448.166,Z 883.974,A 0.000,B 0.000,C 90.000,E1 211.386} C_DIS
LIN {X 0.116,Y -443.924,Z 883.964,A 0.000,B 0.000,C 90.000,E1 209.411} C_DIS
LIN {X 0.121,Y -441.121,Z 883.956,A 0.000,B 0.000,C 90.000,E1 208.103} C_DIS
LIN {X -0.065,Y -436.677,Z 883.945,A 0.000,B 0.000,C 90.000,E1 206.155} C_DIS
LIN {X -0.165,Y -433.225,Z 883.936,A 0.000,B 0.000,C 90.000,E1 204.515} C_DIS
LIN {X -0.127,Y -428.966,Z 883.925,A 0.000,B 0.000,C 90.000,E1 202.514} C_DIS
LIN {X 0.040,Y -424.827,Z 883.914,A 0.000,B 0.000,C 90.000,E1 200.482} C_DIS
LIN {X 0.175,Y -421.465,Z 883.905,A 0.000,B 0.000,C 90.000,E1 198.779} C_DIS
LIN {X -0.250,Y -417.326,Z 883.893,A 0.000,B 0.000,C 90.000,E1 196.804} C_DIS
LIN {X -0.199,Y -411.811,Z 883.878,A 0.000,B 0.000,C 90.000,E1 194.064} C_DIS
LIN {X 0.123,Y -408.526,Z 883.868,A 0.000,B 0.000,C 90.000,E1 192.299} C_DIS
LIN {X -0.122,Y -405.852,Z 883.861,A 0.000,B 0.000,C 90.000,E1 190.950} C_DIS
LIN {X -0.084,Y -402.426,Z 883.851,A 0.000,B 0.000,C 90.000,E1 189.208} C_DIS
LIN {X -0.186,Y -398.171,Z 883.839,A 0.000,B 0.000,C 90.000,E1 187.125} C_DIS
LIN {X 0.180,Y -392.407,Z 883.822,A 0.000,B 0.000,C 90.000,E1 183.898} C_DIS
LIN {X -0.160,Y -387.559,Z 883.804,A 0.000,B 0.000,C 90.000,E1 180.745} C_DIS
LIN {X -0.156,Y -385.448,Z 883.796,A 0.000,B 0.000,C 90.000,E1 179.312} C_DIS
LIN {X 0.094,Y -382.770,Z 883.786,A 0.000,B 0.000,C 90.000,E1 177.478} C_DIS
LIN {X 0.024,Y -380.540,Z 883.778,A 0.000,B 0.000,C 90.000,E1 176.045} C_DIS
LIN {X -0.033,Y -377.005,Z 883.764,A 0.000,B 0.000,C 90.000,E1 173.514} C_DIS
LIN {X -0.084,Y -375.390,Z 883.756,A 0.000,B 0.000,C 90.000,E1 172.064} C_DIS
LIN {X 0.107,Y -374.359,Z 883.746,A 0.000,B 0.000,C 90.000,E1 170.208} C_DIS
LIN {X -0.119,Y -374.364,Z 883.742,A 0.000,B 0.000,C 90.000,E1 169.511} C_DIS
LIN {X 0.020,Y -374.696,Z 883.738,A 0.000,B 0.000,C 90.000,E1 168.757} C_DIS
LIN {X -0.134,Y -375.527,Z 883.734,A 0.000,B 0.000,C 90.000,E1 168.049} C_DIS
LIN {X 0.104,Y -376.513,Z 883.730,A 0.000,B 0.000,C 90.000,E1 167.465} C_DIS
LIN {X -0.093,Y -378.234,Z 883.727,A 0.000,B 0.000,C 90.000,E1 166.881} C_DIS
LIN {X 0.154,Y -381.135,Z 883.723,A 0.000,B 0.000,C 90.000,E1 166.117} C_DIS
LIN {X 0.149,Y -382.038,Z 883.722,A 0.000,B 0.000,C 90.000,E1 165.936} C_DIS
LIN {X 0.149,Y -383.202,Z 883.721,A 0.000,B 0.000,C 90.000,E1 165.755} C_DIS
LIN {X 0.162,Y -387.478,Z 883.718,A 0.000,B 0.000,C 90.000,E1 165.227} C_DIS
LIN {X 0.195,Y -389.211,Z 883.717,A 0.000,B 0.000,C 90.000,E1 165.046} C_DIS
LIN {X 0.034,Y -394.583,Z 883.715,A 0.000,B 0.000,C 90.000,E1 164.629} C_DIS
LIN {X 0.087,Y -405.952,Z 883.711,A 0.000,B 0.000,C 90.000,E1 163.976} C_DIS
LIN {X -0.193,Y -415.944,Z 883.708,A 0.000,B 0.000,C 90.000,E1 163.504} C_DIS
LIN {X 0.049,Y -422.421,Z 883.706,A 0.000,B 0.000,C 90.000,E1 163.087} C_DIS
LIN {X 0.244,Y -431.772,Z 883.703,A 0.000,B 0.000,C 90.000,E1 162.417} C_DIS
LIN {X -0.154,Y -438.201,Z 883.700,A 0.000,B 0.000,C 90.000,E1 162.000} C_DIS
LIN {X 0.111,Y -448.751,Z 883.695,A 0.000,B 0.000,C 90.000,E1 161.094} C_DIS
LIN {X -0.104,Y -453.130,Z 883.693,A 0.000,B 0.000,C 90.000,E1 160.732} C_DIS
LIN {X 0.168,Y -460.503,Z 883.689,A 0.000,B 0.000,C 90.000,E1 160.007} C_DIS
LIN {X -0.112,Y -464.799,Z 883.687,A 0.000,B 0.000,C 90.000,E1 159.625} C_DIS
LIN {X 0.073,Y -470.360,Z 883.684,A 0.000,B 0.000,C 90.000,E1 159.028} C_DIS
LIN {X -0.055,Y -478.631,Z 883.679,A 0.000,B 0.000,C 90.000,E1 158.156} C_DIS
LIN {X -0.151,Y -485.047,Z 883.674,A 0.000,B 0.000,C 90.000,E1 157.411} C_DIS
LIN {X 0.151,Y -493.744,Z 883.669,A 0.000,B 0.000,C 90.000,E1 156.305} C_DIS
LIN {X 0.110,Y -502.809,Z 883.662,A 0.000,B 0.000,C 90.000,E1 155.101} C_DIS
LIN {X -0.195,Y -507.166,Z 883.658,A 0.000,B 0.000,C 90.000,E1 154.537} C_DIS
LIN {X 0.136,Y -518.448,Z 883.649,A 0.000,B 0.000,C 90.000,E1 152.871} C_DIS
LIN {X 0.150,Y -525.336,Z 883.644,A 0.000,B 0.000,C 90.000,E1 151.847} C_DIS
LIN {X -0.109,Y -532.553,Z 883.637,A 0.000,B 0.000,C 90.000,E1 150.717} C_DIS
LIN {X 0.344,Y -538.516,Z 883.632,A 0.000,B 0.000,C 90.000,E1 149.665} C_DIS
LIN {X 0.145,Y -545.733,Z 883.625,A 0.000,B 0.000,C 90.000,E1 148.408} C_DIS
LIN {X -0.060,Y -554.396,Z 883.616,A 0.000,B 0.000,C 90.000,E1 146.882} C_DIS
LIN {X 0.168,Y -561.484,Z 883.608,A 0.000,B 0.000,C 90.000,E1 145.468} C_DIS
LIN {X -0.076,Y -570.354,Z 883.598,A 0.000,B 0.000,C 90.000,E1 143.703} C_DIS
LIN {X 0.328,Y -574.334,Z 883.594,A 0.000,B 0.000,C 90.000,E1 142.844} C_DIS
LIN {X 0.168,Y -583.218,Z 883.583,A 0.000,B 0.000,C 90.000,E1 140.964} C_DIS
LIN {X 0.071,Y -585.604,Z 883.580,A 0.000,B 0.000,C 90.000,E1 140.436} C_DIS
LIN {X 0.124,Y -591.631,Z 883.573,A 0.000,B 0.000,C 90.000,E1 139.094} C_DIS
LIN {X 0.147,Y -595.723,Z 883.568,A 0.000,B 0.000,C 90.000,E1 138.162} C_DIS
LIN {X 0.246,Y -602.451,Z 883.560,A 0.000,B 0.000,C 90.000,E1 136.701} C_DIS
LIN {X 0.111,Y -608.543,Z 883.552,A 0.000,B 0.000,C 90.000,E1 135.405} C_DIS
LIN {X 0.252,Y -613.323,Z 883.547,A 0.000,B 0.000,C 90.000,E1 134.352} C_DIS
LIN {X -0.287,Y -620.112,Z 883.538,A 0.000,B 0.000,C 90.000,E1 132.852} C_DIS
LIN {X -0.101,Y -625.655,Z 883.531,A 0.000,B 0.000,C 90.000,E1 131.553} C_DIS
LIN {X -0.166,Y -629.871,Z 883.525,A 0.000,B 0.000,C 90.000,E1 130.539} C_DIS
LIN {X 0.297,Y -633.986,Z 883.520,A 0.000,B 0.000,C 90.000,E1 129.483} C_DIS
LIN {X -0.082,Y -637.921,Z 883.514,A 0.000,B 0.000,C 90.000,E1 128.508} C_DIS
LIN {X -0.306,Y -641.849,Z 883.508,A 0.000,B 0.000,C 90.000,E1 127.523} C_DIS
LIN {X -0.083,Y -645.737,Z 883.503,A 0.000,B 0.000,C 90.000,E1 126.503} C_DIS
LIN {X 0.237,Y -650.219,Z 883.496,A 0.000,B 0.000,C 90.000,E1 125.231} C_DIS
LIN {X -0.186,Y -653.541,Z 883.490,A 0.000,B 0.000,C 90.000,E1 124.278} C_DIS
LIN {X -0.198,Y -656.625,Z 883.485,A 0.000,B 0.000,C 90.000,E1 123.293} C_DIS
LIN {X -0.090,Y -658.833,Z 883.481,A 0.000,B 0.000,C 90.000,E1 122.546} C_DIS
LIN {X 0.161,Y -661.313,Z 883.475,A 0.000,B 0.000,C 90.000,E1 121.544} C_DIS
LIN {X 0.188,Y -662.440,Z 883.473,A 0.000,B 0.000,C 90.000,E1 121.052} C_DIS
LIN {X -0.285,Y -664.790,Z 883.466,A 0.000,B 0.000,C 90.000,E1 119.873} C_DIS
LIN {X 0.038,Y -666.372,Z 883.460,A 0.000,B 0.000,C 90.000,E1 118.871} C_DIS
LIN {X -0.096,Y -667.468,Z 883.456,A 0.000,B 0.000,C 90.000,E1 118.153} C_DIS
LIN {X 0.095,Y -669.256,Z 883.450,A 0.000,B 0.000,C 90.000,E1 116.924} C_DIS
LIN {X 0.120,Y -669.856,Z 883.447,A 0.000,B 0.000,C 90.000,E1 116.437} C_DIS
LIN {X 0.181,Y -670.817,Z 883.442,A 0.000,B 0.000,C 90.000,E1 115.463} C_DIS
LIN {X -0.209,Y -671.254,Z 883.438,A 0.000,B 0.000,C 90.000,E1 114.771} C_DIS
LIN {X 0.019,Y -671.434,Z 883.434,A 0.000,B 0.000,C 90.000,E1 114.027} C_DIS
LIN {X 0.354,Y -671.196,Z 883.431,A 0.000,B 0.000,C 90.000,E1 113.515} C_DIS
LIN {X -0.197,Y -670.367,Z 883.428,A 0.000,B 0.000,C 90.000,E1 113.078} C_DIS
LIN {X -0.035,Y -669.626,Z 883.427,A 0.000,B 0.000,C 90.000,E1 112.823} C_DIS
LIN {X -0.055,Y -667.515,Z 883.425,A 0.000,B 0.000,C 90.000,E1 112.461} C_DIS
LIN {X 0.021,Y -666.894,Z 883.424,A 0.000,B 0.000,C 90.000,E1 112.333} C_DIS
LIN {X 0.095,Y -666.028,Z 883.423,A 0.000,B 0.000,C 90.000,E1 112.206} C_DIS
LIN {X 0.168,Y -664.671,Z 883.423,A 0.000,B 0.000,C 90.000,E1 112.078} C_DIS
LIN {X 0.073,Y -663.047,Z 883.422,A 0.000,B 0.000,C 90.000,E1 111.972} C_DIS
LIN {X 0.182,Y -660.530,Z 883.421,A 0.000,B 0.000,C 90.000,E1 111.716} C_DIS
LIN {X 0.271,Y -658.857,Z 883.420,A 0.000,B 0.000,C 90.000,E1 111.589} C_DIS
LIN {X 0.038,Y -650.870,Z 883.418,A 0.000,B 0.000,C 90.000,E1 111.280} C_DIS
LIN {X -0.003,Y -647.140,Z 883.418,A 0.000,B 0.000,C 90.000,E1 111.153} C_DIS
LIN {X 0.204,Y -626.858,Z 883.415,A 0.000,B 0.000,C 90.000,E1 110.610} C_DIS
LIN {X 0.125,Y -618.560,Z 883.413,A 0.000,B 0.000,C 90.000,E1 110.375} C_DIS
LIN {X -0.146,Y -610.695,Z 883.412,A 0.000,B 0.000,C 90.000,E1 110.120} C_DIS
LIN {X -0.316,Y -602.025,Z 883.410,A 0.000,B 0.000,C 90.000,E1 109.758} C_DIS
END
